	5:	IF NOT bCheckWrappingSen  (* bIConeFeedingPistonEnd *)    THEN  bQAForwardPistonValve:=FALSE;  bAWrappingConvStart1:=TRUE; bAErrorChkBit:=FALSE;
		step:=step+1; END_IF

	6:	IF  InterLockCounter.CV=1 AND bAConeFeedOver   AND NOT bConeMiss2AtWrapConv THEN
		bA2ndConeReached:=TRUE;
		bAWrappingConvStart1:=FALSE;
		step:=step+1;
		END_IF


	7:	IF NOT bAPauseSeq THEN step:=step+1; END_IF

	8:	 step:=step+1;

	9:	 step:=step+1;

	10:	IF  bAutoModeOn AND NOT bQAWrappingConveyorMotor   AND bA2ndConeReached AND InterLockCounter.CV=1 AND NOT bAConeMissErrorAtWrpConv
		AND NOT bConeMiss2AtWrapConv  THEN
		bQAForwardPistonValve:=TRUE;
		 bAErrorChkBit2:=TRUE;
		bAConeFeedOver:=FALSE;
		step:=step+1;
		END_IF

	11:	IF NOT bAPauseSeq THEN step:=step+1; END_IF

	12:	IF  bAutoModeOn AND bIConeFeedingPistonHome  AND bIForwardPistonEnd  AND NOT bAFwdCylRsError  THEN
		(*bQAForwardPistonValve:=FALSE;*)
		bA2ndConeReached:=FALSE;
		(*bAWrappingConvStart2:=TRUE;  *)
		bAFwdPistonComp2:=TRUE;
		step:=step+1;
		END_IF


	13:	 IF NOT bCheckWrappingSen2 (* bIConeFeedingPistonEnd *) THEN  bQAForwardPistonValve:=FALSE;  bAWrappingConvStart2:=TRUE; bAErrorChkBit2:=FALSE;
		step:=step+1; END_IF
(*-=========================mod need here=======================*)
	14:	IF   bIConeFeedingPistonEnd AND  bAConeFeedOver THEN
		bA3rdConeReached:=TRUE;
		bAWrappingConvStart2:=FALSE;
		step:=step+1;
		END_IF


	15:	IF NOT bAPauseSeq THEN step:=step+1; END_IF

	16:	IF  bAutoModeOn AND NOT bQAWrappingConveyorMotor   AND  bA3rdConeReached  AND  InterLockCounter.CV=2   AND bFwdPistonStartTemp  AND NOT bConeMiss1AtWrapConv  THEN
		bQAForwardPistonValve:=TRUE;
		 bAErrorChkBit3:=TRUE;
		bAConeFeedOver:=FALSE;
		step:=step+1;
		END_IF

	17:	IF NOT bAPauseSeq THEN step:=step+1; END_IF

	18:	IF  bAutoModeOn AND bIConeFeedingPistonHome  AND bIForwardPistonEnd  AND NOT bAFwdCylRsError   THEN

	(*	bQAForwardPistonValve:=FALSE; *)
		bA3rdConeReached:=FALSE;
	(*	bAWrappingConvStart3:=TRUE; *)
		bAFwdPistonComp3:=TRUE;
		step:=step+1;
		END_IF


	19:	IF NOT bAPauseSeq THEN step:=step+1; END_IF


	20:	IF NOT bCheckWrappingSen3 (* bIConeFeedingPistonEnd *) THEN  bQAForwardPistonValve:=FALSE;  bAWrappingConvStart3:=TRUE; bAErrorChkBit3:=FALSE;
		step:=step+1; END_IF



	21:	 IF  bAutoModeOn AND bIForwardPistonHome AND   InterLockCounter.CV=3 OR bAByPassOn    THEN
		InterLockCounter.RESET:=TRUE;
		bAWrappingConvStart3:=FALSE;
		step:=step+1;
		END_IF

	22:	IF NOT bAPauseSeq THEN (* InterLockCounter.RESET:=FALSE ;*) bAByPassOn:=FALSE;  step:=0; END_IF



END_CASE


CASE Step12 OF

	0:	IF R_TRIG_5.Q  THEN Step12:=1; TON_5(IN:=FALSE);  bConutEnable:=FALSE ;END_IF

	1:	IF NOT bQAWrappingConveyorMotor THEN Step12:=2;
		ELSE IF InterLockCounter.CV=2 THEN Step12:=2; END_IF END_IF

	2:	IF  TON_5.Q THEN Step12:=3;
		ELSE IF InterLockCounter.CV=2 AND R_TRIG_1.Q  THEN Step12:=3; END_IF  END_IF

	3:	bConutEnable:=TRUE ; Step12:=4;

	4:	Step12:=0;

END_CASE

R_TRIG_1(CLK:= (  bIWrappingConeDeductionSen), Q=> );
R_TRIG_5(CLK:= (  bWrapConvStarted), Q=> );
TON_5(IN:=bIWrappingConeDeductionSen , PT:=t#0.8s , Q=> , ET=> );

(*IF R_TRIG_1.Q (* bIWrappingConeDeductionSen*)  AND bWrapConvStarted THEN bConutEnable:=TRUE ; ELSE bConutEnable:=FALSE ;END_IF *)

InterLockCounter(
	CU:=bConutEnable ,
	RESET:= ,
	PV:= ,
	Q=> ,
	CV=> );

R_TRIG_2(CLK:=bQAWrappingConveyorMotor , Q=> );

IF R_TRIG_2.Q THEN bWrapConvStarted:=TRUE; END_IF


F_TRIG_1(CLK:= bQAWrappingConveyorMotor, Q=> );

IF F_TRIG_1.Q THEN bWrapConvStarted:=FALSE; END_IF
(*Hanging Logic======*)


IF bAErrorChkBit AND bQAForwardPistonValve  AND  bIWrappingConeDeductionSen  THEN bCheckWrappingSen:=TRUE; END_IF

IF  bWrpConvIntOver AND bSealConvIntOver THEN  bAFwdPistonReady:=TRUE; ELSE 	bAFwdPistonReady:=FALSE; END_IF


IF bAErrorChkBit2 AND  bQAForwardPistonValve AND bIWrappingConeDeductionSen AND (  bIWrappingCone1 OR bIWrappingCone2 OR bIWrappingCone3 ) THEN bCheckWrappingSen2:=TRUE; END_IF


IF bAErrorChkBit3 AND  bQAForwardPistonValve AND bIWrappingConeDeductionSen AND   bIWrappingCone1 AND ( bIWrappingCone2 OR bIWrappingCone3 ) THEN bCheckWrappingSen3:=TRUE; END_IF





IF  NOT bIEmergency OR   bAutoModeOff  OR bStopHmi OR bIMCStop  THEN

bAFirstConeReached:=FALSE;
bQAForwardPistonValve:=FALSE;
bAWrappingConvStart1:=FALSE;
bAFwdPistonComp1:=FALSE;
bA2ndConeReached:=FALSE;
step:=0;
bAWrappingConvStart2:=FALSE;
bAFwdPistonComp2:=FALSE;
bA3rdConeReached:=FALSE;
bAWrappingConvStart3:=FALSE;
bAFwdPistonComp3:=FALSE;
bWrpConvIntOver:=FALSE;
bSealConvIntOver:=FALSE;
InterLockCounter.RESET:=TRUE;

ELSE
InterLockCounter.RESET:=FALSE;

END_IF

IF bErrorReset  AND bCheckWrappingSen AND NOT  bIWrappingConeDeductionSen THEN bAErrorChkBit:=FALSE;  bCheckWrappingSen:=FALSE;WrapConeSenDetMes:=''; InterLockCounter.RESET:=TRUE; ELSE InterLockCounter.RESET:=FALSE;END_IF
IF bCheckWrappingSen THEN  WrapConeSenDetMes:='Wrapping Cone Home Sensor Error';END_IF



IF bErrorReset  AND bCheckWrappingSen2 AND NOT  bIWrappingCone1 AND NOT   bIWrappingCone2 AND NOT bIWrappingCone3  THEN bAErrorChkBit2:=FALSE;  bCheckWrappingSen2:=FALSE;WrapConeSenDetMes:=''; END_IF
IF bCheckWrappingSen2 THEN  WrapConeSenDetMes:='Wrapping Cone Sensor Error';END_IF


IF bErrorReset  AND bCheckWrappingSen3 AND NOT   bIWrappingCone2 AND NOT bIWrappingCone3  THEN bAErrorChkBit3:=FALSE;  bCheckWrappingSen3:=FALSE;WrapConeSenDetMes:=''; END_IF
IF bCheckWrappingSen3 THEN  WrapConeSenDetMes:='Wrapping Cone Sensor Error';END_IF
END_PROGRAM

(* POU AutoMode/Wrapping_Unit, ST *)
PROGRAM Wrapping_Unit
VAR

	step1: INT;

	R_TRIG_1: R_TRIG;
	Counter1: CTU;
	WrapConvStartDly: TON;
	WrapR_TRIG_1: R_TRIG;
	bAWrappingConvStartAuto2: BOOL;
	WrapR_TRIG_2: R_TRIG;
	WrapConvStartDly2: TON;
	WrapR_TRIG_3: R_TRIG;
	WrapConvStartDly3: TON;
	bAWrappingConvStartAuto3: BOOL;
	WrapR_TRIG_4: R_TRIG;
	bAWrappingConvStartAuto4: BOOL;
	WrapConvStartDly4: TON;
	WrapR_TRIG_5: R_TRIG;
	bAWrappingConvStartAuto5: BOOL;
	WrapConvStartDly5: TON;
	bAWrapConeCyl1: BOOL;
	bAWrapConeCyl123: BOOL;
	bAWrapConeCyl3: BOOL;
	bAWrapConeCyl23: BOOL;
	bASet1Comp: BOOL;
	bASet2Comp: BOOL;
	bASet: BOOL;
	bASet3Comp: BOOL;
	bA3ConeWrapStarted: BOOL;
	bA6thConeWrapStarted: BOOL;
	bA1ConeWrappOver: BOOL;
	bA2ConeWrappOver: BOOL;
	bAll3ConeWrapOver: BOOL;
	bA5ConeWrappOver: BOOL;
	bA6ConeWrappOver: BOOL;
	bA56ConeWrapOver: BOOL;
	bAWrapConeCyl23_1: BOOL;

	bATemp: BOOL;
	baConv2ndStart: BOOL;
	baConv3rdStart: BOOL;
	baConv4thStart: BOOL;
	baConv5thStart: BOOL;
	bASensorMonitorBit1: BOOL;
	bAWrappingCone123FwdCom: BOOL;
	ni: BOOL;
	step2: INT;
	bAWrappingCone3FwdCom: BOOL;
	step3: INT;
	bAWrappingCone23FwdCom: BOOL;
	step4: INT;
	bAWrappingCone23FwdCom1: BOOL;
	bASet4Comp: BOOL;
	WrapR_TRIG_3_23: R_TRIG;
	bAWrappingConvStartAuto3_23: BOOL;
	WrapConvStartDly3_23: TON;
	bAWrapConeCyl23_1_23: BOOL;
	bAWrappingCone23_23FwdCom1: BOOL;
	WrapR_TRIG_6_23: R_TRIG;
	bAWrappingConvStartAuto4_23: BOOL;
	WrapConvStartDly6_23: TON;
	bIWrappingCone: BOOL;

	bAWrapConeCyl123_23: BOOL;
	bAWrappingCone123_23FwdCom: BOOL;

	step5: INT;
	bAConvRunning1: BOOL;
	bAConvRunning2: BOOL;
	TON_1: TON;
	TON_2: TON;
	bANextLayerStarted: BOOL;
	bAConvStartInterlock: BOOL;
	bAFirstConeAtWrapConv: BOOL;
	baConveyerStarted: BOOL;
	RtrigBit1: BOOL;
	R_TRIG_3: R_TRIG;
	bASensorNok: BOOL;
	WrapConvStartDlyOver: BOOL;
	test: R_TRIG;
	WrappingCone1RT: R_TRIG;
	WrappingConvRT: R_TRIG;
	WCS1Sensed: BOOL;
	TON_3: TON;
	WCS1SenseRst1: BOOL;
	TON_6: TON;
	TON_7: TON;
	TON_8: TON;
	TON_9: TON;
	TON_10: TON;
	TimerStartBit: BOOL;
	bConvRunning: BOOL;
	test1THEN: BOOL;
	test1: BOOL;
	bSaelUnitIntOverTemp: BOOL;
	step6: INT;
	step7: INT;
	bWCSStart3_24: BOOL;
	bStopHmitemp: BOOL;
	bWCSHomeSenOk: BOOL;

	WCSCylsHomeRsErr: BOOL;

	bWCSHomeEndOk: BOOL;
	WCSCylsEndRsErr: BOOL;

	bAWrappingConvStartAuto: BOOL;
	bA3Pushed: BOOL;
	bWCSStart3: BOOL;
	bWCSStart2: BOOL;
	RsChkDly: TON;
	bWrapConvStopped2: BOOL;

	bWrapConvStopped3: BOOL;

	bIWrappingFilmTensionChk1: BOOL;
	bIWrappingFilmTensionChk2: BOOL;
	bIWrappingFilmTensionChk3: BOOL;
	R_TRIG1: F_TRIG;
	R_TRIG2: F_TRIG;
	R_TRIG3: F_TRIG;
	Film1Loaded: BOOL;
	Film3Loaded: BOOL;
	Film2Loaded: BOOL;
	FlimNotLoaded: BOOL;
	FlimChkDly: TON;
	Timer1: TON;
	bAWrapFirstStart: BOOL;
	TON2: TON;
	sSheetNotFeeded: STRING;
	F_TRIG1: F_TRIG;
	F_TRIG2: F_TRIG;
	F_TRIG3: F_TRIG;
	WrappConeBitAlert1: BOOL;
	WrappConeBitAlert2: BOOL;
	WrappConeBitAlert3: BOOL;
	bQAWrappingConveyorMotor1Temp: BOOL;
	checkPolySheet1: BOOL;
	bQAWrappingConveyorMotor2Temp: BOOL;
	Timer6: TON;
	bAllignConeErr1: BOOL;
	bQAWrappingConveyorMotor2Temp2: BOOL;
	checkPolySheet2Temp: BOOL;

	Timer3: TON;
END_VAR
(*========================Wrapping Conveyor Logic in auto Mode=================*)

bQAWrappingConveyorMotor:= (bQAWrappingConveyorMotor1 OR bQAWrappingConveyorMotor2 OR bQAWrappingConveyorMotor3 );

(*===================Wrapping Pinston On/Off Logic In Auto Mode==================*)


bQAWrappingChannelPistonValve1:= (bAWrappingCone123OnAuto  );

bQAWrappingChannelPistonValve2:=( bAWrappingCone123OnAuto );

bQAWrappingChannelPistonValve3:=( bAWrappingCone123OnAuto );


(*========================Wrapping Conveyor  Logic for First Cone in auto Mode =================*)

WrapR_TRIG_1(CLK:=bAWrappingConvStart1  , Q=> );

IF bAutoModeOn AND  WrapR_TRIG_1.Q  THEN  bAWrappingConvStartAuto:=TRUE; END_IF

WrapConvStartDly(IN:= bAWrappingConvStartAuto, PT:=t#0.3s , Q=> , ET=> );

(*=====New Added for Cone Detection At Wrapp Conveyor====*)

IF WrapR_TRIG_1.Q   AND (bIWrappingCone1 OR bIWrappingCone2 OR  bIWrappingCone3 OR bIWrappingConeDeductionSen) THEN WrappConeBitAlert1:=TRUE;ELSE WrappConeBitAlert1:=FALSE;END_IF
IF WrappConeBitAlert1 AND bErrorReset THEN WrappConeBitAlert1:=FALSE; END_IF
IF WrapR_TRIG_2.Q   AND (bIWrappingCone1 OR bIWrappingCone2 OR  bIWrappingCone3 OR bIWrappingConeDeductionSen) THEN WrappConeBitAlert2:=TRUE;ELSE WrappConeBitAlert2:=FALSE;END_IF
IF WrappConeBitAlert2 AND bErrorReset THEN WrappConeBitAlert2:=FALSE; END_IF
IF WrapR_TRIG_3.Q   AND (bIWrappingCone1 OR bIWrappingCone2 OR  bIWrappingCone3 OR bIWrappingConeDeductionSen) THEN WrappConeBitAlert3:=TRUE;ELSE WrappConeBitAlert3:=FALSE;END_IF
IF WrappConeBitAlert3 AND bErrorReset THEN WrappConeBitAlert3:=FALSE; END_IF


IF bAutoModeOn AND  WrapConvStartDly.Q (*AND NOT bCheckWrappingSen  bIWrappingConeDeductionSen *)AND bIWrappingChannelPiston1_Home AND bIWrappingChannelPiston2_Home  AND  bAWrapFirstStart AND bIWrappingChannelPiston3_Home(*  AND NOT bIWrappingCone1 AND NOT bIWrappingCone2 AND NOT bIWrappingCone3 *) AND NOT WrappConeBitAlert1 THEN
bQAWrappingConveyorMotor1:=TRUE;
bAWrapConStart:=FALSE;
bA3ConeWrappOverTemp:=FALSE;
END_IF

    (*==========================  Wrapping Sheet Sensing Error=================*)
(*
IF bQAWrappingConveyorMotor1   THEN
bAErrorChkBit:=TRUE;

IF NOT  bCheckWrappingSen    THEN
bAErrorChkBit:=FALSE;
bQAWrappingConveyorMotor1Temp:=TRUE;
bQAWrappingConveyorMotor1:=FALSE;
END_IF
END_IF
*)



IF   bAutoModeOn AND  bIWrappingConeDeductionSen THEN
bQAWrappingConveyorMotor1:=FALSE;
bQAWrappingConveyorMotor1Temp:=FALSE;
END_IF

(*===============Wrapping Conveyor 2nd  Cone  Logic  in auto Mode==================*)

WrapR_TRIG_2(CLK:= ( bAWrappingConvStart2 ) , Q=> );


IF bAutoModeOn AND  WrapR_TRIG_2.Q THEN  bAWrappingConvStartAuto:=FALSE;  bAWrappingConvStartAuto2:=TRUE; END_IF

WrapConvStartDly2(IN:= bAWrappingConvStartAuto2, PT:=t#0.1s , Q=> , ET=> );


IF bAutoModeOn AND  WrapConvStartDly2.Q  AND bIWrappingChannelPiston1_Home AND bIWrappingChannelPiston2_Home AND bIWrappingChannelPiston3_Home AND bIWrappingConeDeductionSen   AND NOT bAWrapCylRsErrorAuto AND NOT bConeMiss1AtWrapConv AND NOT WrappConeBitAlert2 AND NOT bCheckWrappingSen2  THEN
bQAWrappingConveyorMotor2:=TRUE;

bAConvRunning1:=TRUE;

END_IF
(*
   (*==========================  Wrapping Sheet Sensing Error=================*)
IF bQAWrappingConveyorMotor2 THEN
IF bQAWrappingConveyorMotor2 AND   bIWrappingConeDeductionSen  AND( bIWrappingCone1 OR  bIWrappingCone2 OR  bIWrappingCone3 ) THEN
checkPolySheet2:=TRUE;
checkPolySheet2Temp:=TRUE;
ELSE
checkPolySheet2Temp:=TRUE;

END_IF
END_IF



IF checkPolySheet2Temp AND   bIWrappingConeDeductionSen AND NOT  bIWrappingCone1 AND NOT  bIWrappingCone2 AND NOT  bIWrappingCone3 AND NOT checkPolySheet2   THEN

bQAWrappingConveyorMotor2Temp:=TRUE; bQAWrappingConveyorMotor2:=FALSE;
END_IF

*)
(*
IF bQAWrappingConveyorMotor2Temp THEN Timer6(IN:=TRUE , PT:=t#2s , Q=> , ET=> ); END_IF

IF bQAWrappingConveyorMotor2Temp AND Timer6.Q AND NOT bIWrappingConeDeductionSen THEN bAllignConeErr1:=TRUE;
ELSIF bQAWrappingConveyorMotor2Temp AND Timer6.Q AND  bIWrappingConeDeductionSen THEN bQAWrappingConveyorMotor2Temp2:=TRUE; Timer6(IN:=FALSE);
END_IF
*)



IF  bAutoModeOn AND  bIWrappingCone1 AND   bAConvRunning1    THEN
bWrapConvStopped2:=TRUE;
bWrapConvStopped2Temp:=TRUE;
bQAWrappingConveyorMotor2:=FALSE;
bAWrappingConvStartAuto2:=FALSE;
bAConvRunning1:=FALSE;
END_IF
(*================================== this Logic is for Cone Missing at Cone Detection sensor in wrapping Unit==========================*)
IF bAutoModeOn AND bWrapConvStopped2Temp AND TON2.Q    AND bIWrappingConeDeductionSen THEN bFwdPistonStartTemp:=TRUE; bWrapConvStopped2Temp:=FALSE; END_IF
IF bAutoModeOn AND bWrapConvStopped2Temp THEN   TON2(IN:=TRUE , PT:= t#1s, Q=> , ET=> ); ELSE TON2(IN:=FALSE);
END_IF
IF bAutoModeOn AND TON2.Q AND NOT  bIWrappingConeDeductionSen  THEN  bConeMiss1AtWrapConv:=TRUE; END_IF

IF bAutoModeOn AND bConeMiss1AtWrapConv AND bIWrappingConeDeductionSen AND bErrorReset AND bIWrappingCone1  THEN
bConeMiss1AtWrapConv:=FALSE; TON2(IN:=FALSE); END_IF

(*===============Wrapping Conveyor  3rd Cone  Logic  in auto Mode ==================*)

WrapR_TRIG_3(CLK:=bAWrappingConvStart3 , Q=> );


IF bAutoModeOn AND  WrapR_TRIG_3.Q THEN bAWrappingConvStartAuto3:=TRUE;  checkPolySheet2Temp:=FALSE; bWrapConvStopped2:=FALSE;  END_IF

WrapConvStartDly3(IN:= bAWrappingConvStartAuto3, PT:=t#0.1s , Q=> , ET=> );


IF  bAutoModeOn AND WrapConvStartDly3.Q AND bIWrappingChannelPiston1_Home AND bIWrappingChannelPiston2_Home AND bIWrappingChannelPiston3_Home AND bIWrappingConeDeductionSen AND bIWrappingCone1 AND NOT bAWrapCylRsErrorAuto AND NOT WrappConeBitAlert3  AND NOT bCheckWrappingSen3  AND NOT  bWrapConvStopped2Temp THEN
bQAWrappingConveyorMotor3:=TRUE;
bASensorMonitorBit1:=TRUE;
END_IF

IF   bAutoModeOn AND  bASensorMonitorBit1 AND   bIWrappingCone3 AND NOT bIWrappingConeDeductionSen THEN
bQAWrappingConveyorMotor3:=FALSE;
bAWrappingConvStartAuto3:=FALSE;
bASensorMonitorBit1:=FALSE;
bWrapConvStopped3:=TRUE;
END_IF
(* ================== Cone Missing Logic on Wrapping Conveyor===============*)

IF bWrapConvStopped3 THEN Timer1(IN:=TRUE , PT:=t#1s , Q=> , ET=> ); ELSE  Timer1(IN:=FALSE); END_IF


IF bAutoModeOn AND   Timer1.Q  AND bWrapConvStopped3 AND bIWrappingCone1 AND bIWrappingCone2 AND NOT bConeMiss2AtWrapConv THEN  bAWrapConeCyl123:=TRUE;  bWrapConvStopped3:=FALSE;
ELSIF bAutoModeOn AND Timer1.Q  AND( NOT  bIWrappingCone1 OR NOT bIWrappingCone2  ) THEN bConeMiss2AtWrapConv:=TRUE;
END_IF


(* ==================Error Acknlodge for  Cone Missing Logic on Wrapping Conveyor===============*)


 IF bConeMiss2AtWrapConv AND bAutoModeOn AND bErrorReset AND   bIWrappingCone1 AND  bIWrappingCone2 AND  bIWrappingCone3  THEN bConeMiss2AtWrapConv:=FALSE;  bAByPassOn:=TRUE; END_IF





(*===============Wrapping piston 123 on/off logic  ====================*)
CASE step1 OF

	0:	TON_1(IN:= FALSE);
		step1:=step1+1;

	1:	step1:=step1+1;

	2:	IF bAutoModeOn AND  bAWrapConeCyl123  AND  bIWrappingChannelPiston1_Home   AND bIWrappingChannelPiston2_Home AND bIWrappingChannelPiston3_Home
		  AND ( bWCSStart1 OR bWCSStart2  )  AND SealingOk AND NOT bAWrapwait THEN
		TON_1(IN:= TRUE, PT:=T#0.3s , Q=> , ET=> );
		IF TON_1.Q THEN  step1:=step1+1; END_IF
		END_IF

	3:	bWCSStart1:=FALSE;
		bWCSStart2:=FALSE;
		step1:=step1+1;


	4:	IF bISealingBottomPistonHome AND bISealingTopPistonHome AND  NOT bQASealingConveyorMotor AND NOT bAPauseSeq   AND NOT bASealSepXCylRsError
		AND SealingOk THEN
		bAWrappingCone123OnAuto:=TRUE;
		step1:=step1+1;
		END_IF


	5:	RsChkDly(IN:=FALSE);
		step1:=step1+1;

	6:	IF bAWrappingCone123OnAuto AND bIWrappingChannelPiston1_End AND bIWrappingChannelPiston2_End AND bIWrappingChannelPiston3_End
		AND SealingOk AND bAFilmLoaded   AND NOT bAWrappingCylRsError THEN
		bAConvRunning1:=FALSE;
		bAWrappingCone123FwdCom:=TRUE;
		TON_1(IN:= FALSE);
		step1:=step1+2;
		ELSIF  bAWrappingCone123OnAuto AND bIWrappingChannelPiston1_End AND bIWrappingChannelPiston2_End AND bIWrappingChannelPiston3_End AND NOT bAWrappingCylRsError  AND NOT bAFilmLoaded THEN
		bAFlimNotLoaded:=TRUE;
		bAWrappingCone123OnAuto:=FALSE;
		bAWrapConeCyl123:=FALSE;
		bAPolythinSheetError:=TRUE;
		ConeMissAlarm1:='Sheet NOT Feeded';
		step1:=step1+3;
		ELSIF NOT  bIWrappingChannelPiston1_End OR NOT  bIWrappingChannelPiston2_End OR NOT  bIWrappingChannelPiston3_End  AND  bAWrappingCone123OnAuto   (* AND not  bAFilmLoaded AND NOT bAWrappingCylRsError     *) THEN
		RsChkDly(IN:=TRUE , PT:=t#5s , Q=> , ET=> );
		IF RsChkDly.Q THEN bAWrapCylRsErrorAuto:=TRUE;   bAWrappingCone123OnAuto:=FALSE; step1:=step1+1; END_IF

		END_IF

	7:	IF bErrorReset THEN RsChkDly(IN:=FALSE);
		bAWrapCylRsErrorAuto:=FALSE;
		step1:=4;
		END_IF

	8:	 IF bAWrappingCone123FwdCom AND NOT bAPauseSeq  THEN
		bAWrappingCone123OnAuto:=FALSE;
		bAFilmLoaded:=FALSE;
		step1:=step1+2;
		END_IF

	9:	 IF bFilmErrClear THEN sSheetNotFeeded:='';  bAFlimNotLoaded:=FALSE;bAConvRunning1:=FALSE;
		 step1:=step1+1;END_IF

	10:	bAWrapConeCyl123:=FALSE;
		bA3ConeWrappOverTemp:=TRUE;
		step1:=step1+1;

	11:	bFilmErrClear:=FALSE;step1:=step1+1;

	12:	 IF  bIWrappingChannelPiston1_Home   AND bIWrappingChannelPiston2_Home AND bIWrappingChannelPiston3_Home   THEN
		bAWrappingCone123FwdCom:=FALSE; 		bA3ConeWrappOver:=TRUE;
		bA3Pushed:=TRUE;
		step1:=0;
		END_IF


END_CASE




IF bAWrapConStart OR bA3ConeWrappOverTemp THEN bAWrapFirstStart:=TRUE; ELSE bAWrapFirstStart:=FALSE; END_IF



	(*========================== Wrapping Sheet not Feeded Error==================*)

	IF bAWrappingCone123OnAuto AND  F_TRIG1.Q AND NOT bIWrappingChannelPiston1_End   AND NOT Film1Loaded THEN Film1Loaded:=TRUE;   END_IF

	IF bAWrappingCone123OnAuto AND  F_TRIG2.Q  AND NOT bIWrappingChannelPiston2_End AND NOT Film2Loaded    THEN Film2Loaded:=TRUE;  END_IF

	IF bAWrappingCone123OnAuto AND  F_TRIG3.Q  AND NOT bIWrappingChannelPiston3_End AND NOT Film3Loaded  THEN Film3Loaded:=TRUE;  END_IF


F_TRIG1(CLK:=bIWrappingFilmTensionPlate_1 , Q=> );


F_TRIG2(CLK:=bIWrappingFilmTensionPlate_2, Q=> );
(* IF R_TRIG2.Q THEN Film2Loaded:=TRUE; END_IF *)


F_TRIG3(CLK:=bIWrappingFilmTensionPlate_3 , Q=> );
  (*IF R_TRIG3.Q THEN Film3Loaded:=TRUE; END_IF *)


IF  Film1Loaded AND  Film2Loaded AND  Film3Loaded THEN bAFilmLoaded:=TRUE;   Film1Loaded:=FALSE;  Film2Loaded:=FALSE;  Film3Loaded:=FALSE;  END_IF

R_TRIG1(CLK:= bAWrappingCone123OnAuto , Q=> );

IF R_TRIG1.Q THEN Film1Loaded:=FALSE; Film2Loaded:=FALSE; Film3Loaded:=FALSE;  END_IF


IF bAWrappingCone123OnAuto THEN FlimChkDly(IN:=TRUE , PT:=t#5s , Q=> , ET=> ); ELSE FlimChkDly(IN:=FALSE);   END_IF

IF bAPolythinSheetError AND bErrorReset   THEN  bFilmErrClear:=TRUE; bAPolythinSheetError:=FALSE ; ConeMissAlarm1:=''; END_IF

(*=============== Interlock Logic for  2*3 WCS conveyor===================*)




IF bSaelUnitIntOver THEN
bSaelUnitIntOverTemp:=TRUE;
END_IF



CASE step6 OF


0:	IF bSaelUnitIntOverTemp   THEN                             (*========= need to check for reset Logic=    step6:=0    =======*)
	Step6:=Step6+1;
	END_IF

1:	bWCSStart1:=TRUE;
	bAWrapConStart:=TRUE;

	Step6:=Step6+1;

2:	IF  bASealConvEnd1 THEN
	bSaelUnitIntOverTemp:=FALSE;
	Step6:=Step6+1;
	END_IF

3:	bWCSStart2:=TRUE;
	bASealConvEnd1:=FALSE;
	Step6:=2;


END_CASE

IF NOT  bIEmergency OR  bAutoModeOff  OR bStopHmi  OR bIMCStop  THEN
bAWrappingConvStartAuto:=FALSE;
WrapConvStartDly(IN:=FALSE);
bQAWrappingConveyorMotor1:=FALSE;
bAWrappingConvStartAuto2:=FALSE;
WrapConvStartDly2(IN:=FALSE);
bQAWrappingConveyorMotor2:=FALSE;
bAConvRunning1:=FALSE;
bWrapConvStopped2:=FALSE;
bFwdPistonStartTemp:=FALSE;
bAWrapCylRsErrorAuto :=FALSE;
bConeMiss1AtWrapConv:=FALSE;
bAWrappingConvStartAuto3:=FALSE;
WrapConvStartDly3(IN:=FALSE);
bQAWrappingConveyorMotor3:=FALSE;
bASensorMonitorBit1:=FALSE;
bWrapConvStopped3:=FALSE;
Timer1(IN:=FALSE);
bAWrapConeCyl123:=FALSE;
bConeMiss2AtWrapConv:=FALSE;
step1:=0;
step6:=0;
TON_1(IN:= FALSE);
bAWrappingCone123OnAuto:=FALSE;
bAWrappingCone123FwdCom:=FALSE;
RsChkDly(IN:=FALSE);
bA3ConeWrappOver:=FALSE;
bA3Pushed:=FALSE;
bIWrappingFilmTensionChk1:=FALSE;
bIWrappingFilmTensionChk2:=FALSE;
bIWrappingFilmTensionChk3:=FALSE;

END_IF
END_PROGRAM

(* POU AutoMode/Sealing_Unit, ST *)
PROGRAM Sealing_Unit
VAR
	step: INT;
	tA3ConeStartDly: TON;
	tA3ConeSealCompDly: TON;
	test: BOOL;


END_VAR
IF NOT  bIEmergency   OR bStopHmi  OR  bAutoModeOff  OR bIMCStop THEN
	Step:=0;
	bQASealingSeparatorYAxisPistonValve:=FALSE;
	bQASealingTopPistonValve:=FALSE;
	bQASealingSeparatorXAxisPistonValve:=FALSE;
	bA3ConeWrappOver:=FALSE;
	bMManualSealOn:=FALSE;
	tA3ConeStartDly(IN:=FALSE);
	tA3ConeSealCompDly(IN:=FALSE);

END_IF


CASE step OF

	0:	IF bAutoModeOn  THEN
		Step:=step+1;
		END_IF

	1:	step:=step+1;


	2:	IF bAutoModeOn AND  bA3ConeWrappOver   AND NOT bAPauseSeq  THEN
		tA3ConeStartDly(IN:=TRUE , PT:=t#1.5s , Q=> , ET=> );
		IF tA3ConeStartDly.Q THEN  step:=step+1; END_IF
		END_IF

	3:	step:=step+1;

	4:	IF bAutoModeOn AND   bISealingBottomPistonHome  AND bISealingTopPistonHome AND bISealingSeparatorXAxisHome AND bISealingSeparatorYAxisHome AND  NOT bAPauseSeq THEN
		bQASealingSeparatorYAxisPistonValve:=TRUE;
		bASepYAxisRsErrorChkBit:=TRUE;
		tA3ConeSealCompDly(IN:=FALSE);
		step:=step+1;
		END_IF

	5:	 step:=step+1;

	6:	IF bAutoModeOn AND  bISealingSeparatorYAxisEnd AND  NOT bAPauseSeq  AND NOT bASealSepYCylRsError THEN
		tA3ConeStartDly(IN:=FALSE);
		bQASealingTopPistonValve:=TRUE;
		bASepYAxisRsErrorChkBit:=FALSE;
		step:=step+1;
		END_IF

	7:	step:=step+1;

	8:	IF bAutoModeOn AND  bISealingTopPistonEnd AND bISealingBottomPistonEnd  THEN
		tA3ConeSealCompDly(IN:=TRUE, PT:= SealComDlyTemp, Q=> , ET=> );
		IF tA3ConeSealCompDly.Q THEN   step:=step+1; END_IF
		END_IF

	9:	step:=step+1;

	10:	IF bAutoModeOn AND  bISealingTopPistonEnd AND bISealingBottomPistonEnd (*AND  bISealingSeparatorYAxisEnd*) AND  NOT bAPauseSeq  AND NOT bASealTopBotCylRsError  AND NOT bASealSepYCylRsError  THEN
		bQASealingSeparatorXAxisPistonValve:=TRUE;
		(*bASepYAxisRsErrorChkBit1:=TRUE;  *)
		step:=step+1;
		END_IF

	11:	 bASepYAxisRsErrorChkBit1:=FALSE; step:=step+1;

	12:	IF bAutoModeOn AND  bISealingSeparatorXAxisEnd AND  NOT bAPauseSeq  AND NOT bASealSepXCylRsError THEN

		step:=step+1;
		 END_IF

	13:	 step:=step+1;

	14:	bQASealingTopPistonValve:=FALSE;
		bA3ConeWrappOver:=FALSE;
		bA4thWrappOver:=FALSE;
		bA6thConeWrappOver:=FALSE;
		bA8thConeWrappOver:=FALSE;
		bA6ConeWrappOver23:=FALSE;
		bQASealingSeparatorYAxisPistonValve:=FALSE;
		bQASealingSeparatorXAxisPistonValve:=FALSE;
		step:=step+1;

	15:	step:=step+1;

	16:	IF bAutoModeOn AND  bISealingSeparatorXAxisHome AND  bISealingTopPistonHome AND bISealingBottomPistonHome AND bISealingSeparatorYAxisHome  THEN
		step:=step+1;
		END_IF


	17:	step:=step+1;

	18:	step:=step+1;

	19:	 step:=step+1;

	20:	step:=0;



END_CASE

		IF bAutoModeOn AND NOT bA3ConeWrappOver  AND NOT bA4thWrappOver AND NOT bA6thConeWrappOver AND NOT bA8thConeWrappOver
		 AND  bISealingSeparatorXAxisHome AND  bISealingTopPistonHome AND bISealingBottomPistonHome AND bISealingSeparatorYAxisHome  THEN
		SealingOk:=TRUE; ELSE SealingOk:=FALSE;
		END_IF













































(*

(*================Wrapping Conveyor On/Off Logic==========================*)

CASE step OF
	1:	IF SealDelay.Q   AND NOT bIColumnPushPistonHome THEN
		bQAWrappingConveyorMotor:=TRUE;
		END_IF
	2:	IF bIConeCountSensorVal=3 THEN bQAWrappingConveyorMotor:=FALSE; END_IF

	3: 	IF SealDelay.Q  AND NOT bIColumnPushPistonHome   THEN  bQAWrappingConveyorMotor:=TRUE;	END_IF

	4:	IF bIConeCountSensorVal=1 THEN bQAWrappingConveyorMotor:=FALSE; END_IF

	5:	 IF SealDelay.Q   AND NOT bIColumnPushPistonHome   THEN  bQAWrappingConveyorMotor:=TRUE;	END_IF

	6:	IF bIConeCountSensorVal=2 THEN bQAWrappingConveyorMotor:=FALSE; END_IF


	7:	 IF SealDelay.Q   AND NOT bIColumnPushPistonHome   THEN  bQAWrappingConveyorMotor:=TRUE;	END_IF

	8:	IF bIConeCountSensorVal=2 THEN bQAWrappingConveyorMotor:=FALSE; END_IF


	9:	step:=0;


END_CASE

*)







(*


		IF bAutoModeOn AND  bAWrapConeCyl123 AND bIWrappingChannelPiston1_Home   AND bIWrappingChannelPiston2_Home AND bIWrappingChannelPiston3_Home    THEN
		bAWrappingCone123OnAuto:=TRUE;

		END_IF

		IF  bAutoModeOn AND  bIWrappingChannelPiston1_End AND bIWrappingChannelPiston2_End AND bIWrappingChannelPiston3_End   THEN
		bAWrappingCone123OnAuto:=FALSE;
		bAWrapConeCyl123:=FALSE;


		END_IF

	IF  bAutoModeOn AND  bAWrappingCone123OnAuto  THEN
		bA3ConeWrapStarted:=TRUE;
	END_IF

IF  bA3ConeWrapStarted AND bIWrappingChannelPiston1_End THEN
bA1ConeWrappOver:=TRUE;END_IF

 IF bA3ConeWrapStarted AND bIWrappingChannelPiston2_End THEN
bA2ConeWrappOver:=TRUE;
END_IF

IF bA3ConeWrapStarted AND  bIWrappingChannelPiston3_End THEN
bA3ConeWrappOver:=TRUE;
END_IF


IF bA1ConeWrappOver AND bA2ConeWrappOver AND bA3ConeWrappOver  THEN
bAll3ConeWrapOver:=TRUE;
 bASet1Comp:=TRUE;
END_IF


*)
END_PROGRAM

(* POU AutoMode/Sealing_Conveyor, ST *)
PROGRAM Sealing_Conveyor
VAR

	bA3ConeSealStarted23: BOOL;
	bQASealingConveyor2: BOOL;
	ConvStopDly1_23: TON;
	bA3ConeSealComp23: BOOL;
	step1: INT;
	(*CTU_1: CTU;*)
	bAConeCountSenEnable1: BOOL;
	bA6thConeSealStarted23: BOOL;
	bA6thConeSealComp23: BOOL;
	ConvStopDly2_23: TON;
	step2: INT;
	step3: INT;
	bSealConvIntOverTemp: BOOL;
	bStopHmitemp: BOOL;
	ConeMissErr_1: BOOL;

	ConeMissErr_2: BOOL;
	test: BOOL;
	bA3COneCrossed: BOOL;
	bSealConvStart3: BOOL;
	bSealConvStart1: BOOL;
	TON1: TON;
	Timer1: TON;
	Timer2: TON;

	Timer3: TON;
	bConeMissBit2: BOOL;
	bConeMissBit3: BOOL;
	bConeMissBit1: BOOL;
	Timer4: TON;
	bConeMissBit: BOOL;
	ConeChkDly: TON;
	SealConeMiss: STRING;
	bQASealingConveyor3: BOOL;
	bAConeMissAtSealConv2: BOOL;
	bA3ConeSealComp23Temp: BOOL;
	bTemp: BOOL;

END_VAR
bQASealingConveyorMotor:= bQASealingConveyor1 OR bQASealingConveyor2 OR bQASealingConveyor3 ;


CASE step1 OF

	0:	IF bAutoModeOn  AND   bA3ConeWrappOver AND bQASealingSeparatorYAxisPistonValve  THEN
		CTU_1.RESET:=TRUE;
		TON1(IN:=FALSE);
		bA3ConeSealStarted23:=TRUE;
		ConvStopDly1_23(IN:=FALSE);
		step1:=step1+1;
		END_IF
	1:	IF NOT bAPauseSeq THEN step1:=step1+1; END_IF


	2:	IF bAutoModeOn  AND  bA3ConeSealStarted23 AND bISealingSeparatorXAxisEnd THEN
		bA3ConeSealComp23:=TRUE;
		CTU_1.RESET:=FALSE;
		step1:=step1+1;
		END_IF

	3:	step1:=step1+1;

	4:	IF bAutoModeOn AND   bA3ConeSealComp23Temp  AND   NOT bAPauseSeq    AND NOT bASealSepXCylRsError THEN
		bQASealingConveyor1:=TRUE;
		step1:=step1+1;
		END_IF

	5:	 TON1(IN:=FALSE); step1:=step1+1;


	6:	IF CTU_1.CV>=3 THEN
		bSealConvStart1:=FALSE;
		bSealConvStart3:=FALSE;
		bA3ConeSealComp23Temp:=FALSE;
		bA3ConeSealStarted23:=FALSE;
		bA3COneCrossed:=TRUE;
		TON1(IN:=TRUE, PT:=  t#1s, Q=> , ET=> );
		IF TON1.Q THEN  CTU_1.RESET:=TRUE; step1:=step1+1; END_IF
		END_IF

	7:	bQASealingConveyor1:=FALSE;
		bQASealingConveyor2:=FALSE;
		bQASealingConveyor3:=FALSE;
		bASealConvEnd1:=TRUE;
		CTU_1.RESET:=FALSE;
		TON1(IN:=FALSE);

		step1:=0;



END_CASE

IF NOT bQASealingConveyorMotor AND bIConeCountSensor  THEN bAWrapwait:=TRUE;ELSE bAWrapwait:=FALSE;END_IF

IF bA3ConeSealComp23 THEN  bA3ConeSealComp23Temp:=TRUE;  bA3ConeSealComp23:=FALSE; END_IF


IF bQASealingConveyorMotor AND bIConeCountSensor  THEN
bAConeCountSenEnable1:=TRUE;
ELSE
bAConeCountSenEnable1:=FALSE;
END_IF

CTU_1(
	CU:=bAConeCountSenEnable1 ,
	RESET:= ,
	PV:=3 ,
	Q=> ,
	CV=> );

IF CTU_1.CV<>3 AND (bQASealingConveyor1 OR bQASealingConveyor2 OR bQASealingConveyor3 )THEN
(*ConeMissbit:=TRUE;*)
ConeChkDly(IN:= TRUE , PT:=t#7s , Q=> , ET=> );
ELSE
ConeChkDly(IN:= FALSE);
END_IF


(*
CASE SealingStep OF



	0:	Timer1(IN:=FALSE);
		Timer2(IN:=FALSE);
		Timer3(IN:=FALSE);
		SealingStep:=SealingStep+1;

	1:	IF  ConeMissbit  THEN
		Timer1(IN:=TRUE , PT:=t#2s , Q=> , ET=> );
		IF NOT Timer1.Q  AND (CTU_1.CV ) = 1 THEN SealingStep:=SealingStep+1;
		ELSIF  Timer1.Q	 AND (CTU_1.CV)<>1 THEN  SealingStep:=3;
		END_IF
		END_IF

	2:	IF (CTU_1.CV)=1 THEN
		SealingStep:=SealingStep+2;
		END_IF

	3:	IF  (CTU_1.CV)<>1 THEN
		bConeMissBit1:=TRUE;
		AlarmMessg:='One Cone  Missing From Sealing Conveyor';
		SealingStep:=11;
		ELSIF (CTU_1.CV) = 1  THEN
		AlarmMessg:='';
		SealingStep:=SealingStep+1;
		END_IF


	4:	Timer2(IN:=TRUE , PT:=t#2s , Q=> , ET=> );
		IF NOT Timer2.Q  AND (CTU_1.CV ) = 2 THEN SealingStep:=SealingStep+1;
		ELSIF  Timer2.Q	 AND (CTU_1.CV)<>2 THEN  SealingStep:=6; END_IF


	5:	IF (CTU_1.CV)=2 THEN
		SealingStep:=SealingStep+2; END_IF




	6:	IF  (CTU_1.CV)<>2 THEN
		bConeMissBit2:=TRUE;
		AlarmMessg:='Two Cone  Missing From Sealing Conveyor';
		SealingStep:=11;
		ELSIF (CTU_1.CV) = 2  THEN
		AlarmMessg:='';
		SealingStep:=SealingStep+1;

		END_IF

	7:	Timer3(IN:=TRUE , PT:=t#2s , Q=> , ET=> );
		IF NOT Timer3.Q AND  NOT bAPauseSeq  AND (CTU_1.CV ) =3 THEN SealingStep:=SealingStep+1;
		ELSIF  Timer3.Q AND  NOT bAPauseSeq	 AND (CTU_1.CV)<>3 THEN  SealingStep:=9; END_IF

	8:	IF (CTU_1.CV)=3 THEN
		SealingStep:=10;
		END_IF

	9:	IF (CTU_1.CV) <> 3  THEN
		bConeMissBit3:=TRUE;
		AlarmMessg:='One Cone  Missing From Sealing Conveyor';
		SealingStep:=11;
		ELSIF (CTU_1.CV) = 3  THEN
		AlarmMessg:='';
		SealingStep:=SealingStep+1;
		END_IF


	10:	IF (CTU_1.CV)=0 THEN
		ConeMissbit:=FALSE;
		Timer3(IN:=FALSE);
		Timer2(IN:=FALSE);
		Timer1(IN:=FALSE);
		SealingStep:=0;
		END_IF

	11:	Timer4(IN:=TRUE , PT:= t#3m, Q=> , ET=> );
		IF bConeMissBit  AND  (CTU_1.CV)=1  AND  Timer4.Q THEN(* bAPauseEnable:=TRUE; *)  bQASealingConveyor1:=FALSE;  Step1:=4;  SealingStep:=7;
		ELSIF bConeMissBit  AND  (CTU_1.CV)=2  AND  Timer4.Q THEN (*bAPauseEnable:=TRUE; *) bQASealingConveyor1:=FALSE;  Step1:=4;  SealingStep:=7;
		END_IF

END_CASE




IF bQASealingConveyor1_23 AND CTU_AlarmOnly.CV =3  THEN  bCountLock1:=TRUE; END_IF

IF bQASealingConveyor5_23 AND CTU_AlarmOnly.CV =3  THEN  bCountLock5:=TRUE; END_IF

IF bQASealingConveyor6_23 AND CTU_AlarmOnly.CV =3  THEN  bCountLock6:=TRUE; END_IF


IF bQASealingConveyor2_23 AND CTU_AlarmOnly.CV =6  THEN  bCountLock2:=TRUE; END_IF


IF bQASealingConveyor3_23 AND CTU_AlarmOnly.CV =6  THEN  bCountLock3:=TRUE; END_IF


IF bQASealingConveyor4_23 AND CTU_AlarmOnly.CV =6  THEN  bCountLock4:=TRUE; END_IF


 IF bCountLock1 OR bCountLock2 OR  bCountLock3 OR bCountLock4 OR  bCountLock5 OR bCountLock6 THEN bCountLock:=TRUE; ELSE bCountLock:=FALSE; END_IF
*)


IF bQASealingConveyor1  AND  ConeChkDly.Q   AND   CTU_1.CV<>3  THEN bAConeMissAtSealConv:=TRUE; AlarmMessg:=' Cone  Missing From Sealing Conveyor';  bQASealingConveyor1:=FALSE;  END_IF




IF bAConeMissAtSealConv AND bErrorReset THEN bQASealingConveyor2:=TRUE;  Step1:=5;    AlarmMessg:=''; bAConeMissAtSealConv:=FALSE; END_IF

IF bQASealingConveyor2  AND  ConeChkDly.Q   AND CTU_1.CV<>3   THEN bAConeMissAtSealConv2:=TRUE; AlarmMessg:=' Cone  Missing From Sealing Conveyor';  bQASealingConveyor2:=FALSE;  END_IF

IF bAConeMissAtSealConv2 AND bErrorReset THEN bQASealingConveyor3:=TRUE;  Step1:=5;  ConeChkDly(IN:= FALSE);  AlarmMessg:=''; bAConeMissAtSealConv2:=FALSE; END_IF

IF bQASealingConveyor3 AND ConeChkDly.Q  AND CTU_1.CV<>3 THEN bQASealingConveyor3:=FALSE; bTemp:=TRUE;  AlarmMessg:=' Cone  Missing From Sealing Conveyor'; END_IF

IF bTemp  AND bErrorReset THEN
Step1:=4;  ConeChkDly(IN:= FALSE); bTemp:=FALSE;
END_IF



IF bAConeMissAtSealConv OR bAConeMissAtSealConv2 THEN bAConeMissAtSealConv:=TRUE; ELSE  bAConeMissAtSealConv:=FALSE; END_IF



IF NOT  bIEmergency OR  bAutoModeOff  OR bStopHmi OR bIMCStop  THEN
step1:=0;
bA3ConeSealStarted23:=FALSE;
ConvStopDly1_23(IN:=FALSE);
bA3ConeSealComp23:=FALSE;
bQASealingConveyor1:=FALSE;
bQASealingConveyor2:=FALSE;
bQASealingConveyor3:=FALSE;
bAConeMissAtSealConv:=FALSE;
bAConeMissAtSealConv2:=FALSE;
bAConeMissAtSealConv:=FALSE;
CTU_1.RESET:=TRUE;
bAConeCountSenEnable1:=FALSE;
TON1(IN:=FALSE);
ELSE

CTU_1.RESET:=FALSE;

END_IF
END_PROGRAM

(* POU WeightCalc, ST *)
PROGRAM WeightCalc
VAR
	CounterA: CTU;
	R_TRIG_1: R_TRIG;
	CounterB: CTU;
	R_TRIG_2: R_TRIG;
	R_TRIG_3: R_TRIG;

	ConeCountEnable: BOOL;
	InterLockCounterStartTimer: TON;
	TON_3: TON;
	tResetTiner: TON;
	WCPReadyTemp1: BOOL;
	WCPReadyTemp2: BOOL;
	Det: WORD;
	BreadTemp: BOOL;
	ADSREAD_1: ADSREAD;
	SwithOnButtton: BOOL;
	axis1: BOOL;
	InterLockCounterRESET: BOOL;
	RstStep: INT;
	bStopTiltUnit: BOOL;
	rRetUnitTolMax: REAL;
	rRetUnitTolMin: REAL;
	rRetUnitAWeightok: BOOL;

	TON_4: TON;
	rRetUnitAWeightempt: REAL;
	rRetUnitAWeighttemp: REAL;
	TON_5: TON;
	rRetUnitBWeightok: BOOL;
	TON_6: TON;
	TON_7: TON;
	rGrossWtTolMax: REAL;
	rGrossWtTolMin: REAL;
	TON_8: TON;
	bGrossWieghtOkTemp: BOOL;

	Timer1: TON;
	Timer2: TON;
	bMonitor: BOOL;
	bStartBlinker: BOOL;
	bStartConeFeedConvInBypass: BOOL;
	rRetUnitAWeightNok: BOOL;
	rRetUnitBWeightNok: BOOL;
	iACounterB_PV: INT;
	iACounterA_PV: INT;
	i: INT;

	UnitBWeightBit: BOOL;
	UnitAWeightBit: BOOL;
	weightCheck: INT;
	Timer_3: TON;
	Weight3Move: BOOL;
	var_4: REAL;
	weightCheck1: INT;
	Weight4Move: BOOL;
	Timer_4: TON;
	Weight2Move: BOOL;
	var_2: REAL;
	var_3: REAL;
	Weight1Move: BOOL;
END_VAR
(*===========Reterival unit weight ok and not ok Logic UNIT-A=================*)

(*==== Weight Max & Min Tolerance Setting==========*)

rRetUnitTolMax:= (DFLTNETWT_DIS + NETWTTOL_DIS);

	IF negativetolerance AND bAutoModeOn THEN
	rRetUnitTolMin:= (DFLTNETWT_DIS - NETWTTOL_DIS);
	ELSIF NOT negativetolerance THEN rRetUnitTolMin:= (DFLTNETWT_DIS);
	END_IF
IF rRetUnitAWeight  <= rRetUnitTolMax AND rRetUnitAWeight >=rRetUnitTolMin THEN
rRetUnitAWeightok:=TRUE;
ELSE
rRetUnitAWeightok:=FALSE;
END_IF

IF TON_5.Q   THEN bQAUnitAWeightOkLamp:=TRUE; END_IF


(*
ELSIF Timer1.Q THEN bQAUnitA_LiftPistonValve:=TRUE; ELSE  bQAUnitA_LiftPistonValve:=TRUE; END_IF
IF  bUnitARowStopperStarted  THEN bStartBlinker:=TRUE; ELSE   bStartBlinker:=FALSE;


Timer1(IN:=(bStartBlinker AND NOT Timer2.Q)  , PT:=t#50ms , Q=> , ET=> );

Timer2(IN:=Timer1.Q , PT:=t#50ms , Q=> , ET=> );
*)



(*=========== Unit A Start after wieght ok logic=================*)

IF bIUnitA_StartPB  AND bQAUnitAWeightOkLamp AND bAutoModeOn AND NOT bStartConeFeedConvInBypass THEN  bRetUnitAStart:=TRUE; ELSE bRetUnitAStart:=FALSE;  END_IF





(*============Weight stabilization time======================*)


IF rRetUnitAWeightok THEN TON_4(IN:=TRUE , PT:=t#2s , Q=> , ET=> ); ELSE  TON_4(IN:=FALSE); END_IF

(*============== WEIGHT NOT OK DEFINE TIME ( TON_5)=================*)

IF TON_4.Q THEN TON_5(IN:=TRUE , PT:=t#0.5s , Q=> , ET=> ); ELSE TON_5(IN:=FALSE); END_IF

IF bAutoModeOn AND bIUnitA_RowStopperHome AND NOT rRetUnitAWeightok THEN rRetUnitAWeightNok:=TRUE;  bQAUnitAWeightOkLamp:=FALSE;  ELSE rRetUnitAWeightNok:=FALSE;   END_IF
(*
  IF rRetUnitAWeightNok THEN bRetUnitAStart:=FALSE; END_IF
*)


(*===============weight not ok Indicator on logic====================*)

IF rRetUnitAWeightNok THEN bQAUnitAWeightNokLamp:=TRUE; ELSE  bQAUnitAWeightNokLamp:=FALSE;  END_IF


(*================ Weight ok feedback to Auto Logic=============*)

IF  rRetUnitAWeightok THEN bAUnitAWeighOk:=TRUE;  ELSE bAUnitAWeighOk:=FALSE; END_IF


(*===========Reterival unit weight ok and not ok Logic UNIT-B =================*)



IF rRetUnitBWeight  <= rRetUnitTolMax AND rRetUnitBWeight >=rRetUnitTolMin THEN
rRetUnitBWeightok:=TRUE;
ELSE
rRetUnitBWeightok:=FALSE;
END_IF

IF TON_7.Q THEN bQAUnitBWeightOkLamp:=TRUE; ELSE  bQAUnitBWeightOkLamp:=FALSE;  END_IF




(*=========== Unit B Start after wieght ok logic=================*)

IF bIUnitB_StartPB  AND bQAUnitBWeightOkLamp AND bAutoModeOn  AND NOT bStartConeFeedConvInBypass  THEN  bRetUnitBStart:=TRUE; ELSE bRetUnitBStart:=FALSE; END_IF


(*============Weight stabilization time======================*)


IF rRetUnitBWeightok THEN TON_6(IN:=TRUE , PT:=t#2s , Q=> , ET=> ); ELSE  TON_6(IN:=FALSE); END_IF

(*============== WEIGHT NOT OK DEFINE TIME ( TON_5)=================*)

IF TON_6.Q THEN TON_7(IN:=TRUE , PT:=t#0.5s , Q=> , ET=> ); ELSE TON_7(IN:=FALSE); END_IF

IF bAutoModeOn  AND bIUnitB_RowStopperHome AND NOT rRetUnitBWeightok THEN rRetUnitBWeightNok:=TRUE; ELSE rRetUnitBWeightNok:=FALSE;   END_IF
(*
  IF rRetUnitBWeightNok THEN bRetUnitBStart:=FALSE; END_IF
*)


(*===============weight not ok Indicator on logic====================*)


IF rRetUnitBWeightNok THEN bQAUnitBWeightNokLamp:=TRUE; ELSE  bQAUnitBWeightNokLamp:=FALSE;  END_IF


(*================ Weight ok feedback to Auto Logic=============*)

IF  rRetUnitBWeightok THEN bAUnitBWeighOk:=TRUE; ELSE bAUnitBWeighOk:=FALSE;  END_IF




(*============================================================================================================================================================*)



(*===================UnitA Cone Count Logic================*)

CounterA(
	CU:=bIUnitAConeCrossing ,
	RESET:=R_TRIG_1.Q ,
	PV:=iACounterA_PV ,
	Q=> ,
	CV=> );



(*===================UnitB Cone Count Logic================*)

CounterB(
	CU:=bIUnitBConeCrossing ,
	RESET:=R_TRIG_2.Q ,
	PV:=iACounterB_PV ,
	Q=> ,
	CV=> );





IF bRetUnitAStart AND NOT bRetUnitBStart  (*AND NOT UnitBWeightBit *)THEN UnitAWeightBit:=TRUE; var_1:=rRetUnitAWeight; END_IF
IF bRetUnitBStart AND NOT bRetUnitAStart (*AND NOT UnitAWeightBit*)  THEN UnitBWeightBit:=TRUE; var_2:=rRetUnitBWeight; END_IF

CASE  weightCheck OF


	0:	IF  UnitAWeightBit AND NOT UnitBWeightBit THEN
		Weight1Move:=TRUE;
		weightCheck:=1;END_IF

	1:	IF  Weight1Move AND NOT Weight3Move THEN
		var_3:=var_1;
		Weight3Move:=TRUE;
		Weight1Move:=FALSE;

		weightCheck:=2;END_IF

	2:	IF  CycleComplete AND Weight3Move THEN
		 var_5:=var_3;
		ReportPrint:=TRUE;

		weightCheck:=3;END_IF

	3: 	IF Weight3Move THEN Timer_3(IN:=TRUE , PT:= T#1s , Q=> , ET=> );
		IF Timer_3.Q THEN Weight3Move:=FALSE; UnitAWeightBit:=FALSE;Timer_3(IN:=FALSE);
		weightCheck:=0;END_IF END_IF

END_CASE

CASE  weightCheck1 OF

	0:	IF  UnitBWeightBit AND NOT UnitAWeightBit THEN
		Weight2Move:=TRUE;
		weightCheck1:=1;END_IF

	1:	IF  Weight2Move AND NOT Weight4Move THEN
		var_4:=var_2;
		Weight4Move:=TRUE;
		Weight2Move:=FALSE;

		weightCheck1:=2;END_IF

	2:	IF  CycleComplete1 AND Weight4Move  THEN
		var_5:=var_4;
		ReportPrint:=TRUE;

		weightCheck1:=3;END_IF

	3: 	IF Weight4Move THEN Timer_4(IN:=TRUE , PT:= T#1s , Q=> , ET=> );
		IF Timer_4.Q THEN Weight4Move:=FALSE;UnitBWeightBit:=FALSE; Timer_4(IN:=FALSE);
		weightCheck1:=0;END_IF END_IF

END_CASE


IF  NOT bIEmergency OR   bAutoModeOff  OR bStopHmi OR bIMCStop  THEN

weightCheck1:=0;
weightCheck:=0;
Weight4Move:=FALSE;
Weight2Move:=FALSE;
Weight3Move:=FALSE;
 UnitAWeightBit:=FALSE;
Timer_3(IN:=FALSE);
Weight1Move:=FALSE;
UnitAWeightBit:=FALSE;
UnitBWeightBit:=FALSE;
END_IF
END_PROGRAM

(* POU Startup/INT_All, ST *)
PROGRAM INT_All
VAR
	bCartonOnConv: BOOL;
	bWrpConvIntOverTemp: BOOL;
	bSealConvIntOverTemp: BOOL;
	bAInializeStartedtenp: BOOL;
	bStopInt: BOOL;

	F_TRIG_1: F_TRIG;

END_VAR
IF bInitializeHmi AND bAMcStartInAuto  AND bAutoModeOn (*AND bMCStartInAuto   *) AND NOT   bAInializeStarted    AND NOT bInterlockInitial_2 THEN
bAInitializeSeq:=TRUE;
bAInializeStarted:=TRUE;
bIntialAckBit:=TRUE;
bInterlockInitial_2:=TRUE;
bUnitBReadInt:=TRUE;
END_IF

blink();

WrapConvRst();


SealingConvRst();


SealingUnitRst();



IF  bWrpConvIntOver   AND bSealConvIntOver THEN bAInializeStarted:=FALSE ; bIntialAckBit:=FALSE;END_IF

IF bStopHmi OR bIMCStop  AND bAutoModeOn   THEN bAStop :=TRUE;  bWrpConvIntOver:=FALSE; bSealConvIntOver:=FALSE;  bAMcReady:=FALSE; END_IF

IF( bStopHmi OR bIMCStop)  AND bAutoModeOn AND NOT  bIEmergency THEN bInterlockInitial_2:=FALSE; bUnitBReadInt:=FALSE;END_IF


F_TRIG_1(CLK:= bAInializeStarted, Q=> );

IF F_TRIG_1.Q  AND bAutoModeOn AND   bWrpConvIntOver   AND bSealConvIntOver THEN   bAMcReady:=TRUE; END_IF


IF bAMcReady AND bAutoModeOn AND (bRetUnitAStart OR bRetUnitBStart  ) THEN bAMcRunninig:=TRUE;  bAMcReady:=FALSE; END_IF

(* IF NOT bIEmergency OR bIMCStop   OR bInitializeHmi  THEN bStopInt:=TRUE; ELSE bStopInt:=FALSE; END_IF  *)

(*
AlarmList();
*)


(*
(*=============FULL CARTON CONVEYOR INITIALIZE LOGIC==========*)

	IF    bICartonPosition1 OR  bICartonPosition2 OR  bICartonPosition3  THEN bCartonOnConv:=TRUE; ELSE  bCartonOnConv:=FALSE;  END_IF

	IF 	bAInitializeSeq  AND  bCartonOnConv   AND bAutoModeOn  THEN
	sCartonConvStatus:='Clear the Cone on Carton Conveyor';
	ELSIF 	bAInitializeSeq AND NOT bCartonOnConv AND bAutoModeOn THEN
	bClearConeInt:=TRUE;
	bCartonOnConv:=FALSE;
	sCartonConvStatus:='';
	END_IF
*)
END_PROGRAM

(* POU Startup/blink, CFC *)
PROGRAM blink
VAR
	timer1: TON;
	timer2: TON;
END_VAR
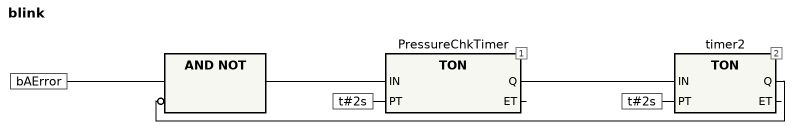
_CFC_ (* Continuous Function Chart, elements in execution order *)
#0 AND NOT(bAError, NOT #2.Q)
#1 PressureChkTimer:TON(IN: #0, PT: t#2s)
#2 timer2:TON(IN: #1.Q, PT: t#2s)
_END_CFC_
END_PROGRAM

(* POU Startup/WrapConvRst, ST *)
PROGRAM WrapConvRst
VAR
	step: INT;
	bConeAtWrppingConveyor1: BOOL;
	TON_1: TON;
	bConePresent: BOOL;
	bAResetHmitemp: BOOL;

	ConeOnWrapConveyAck: BOOL;
END_VAR
IF NOT  bIEmergency OR bStopHmi  OR bAutoModeOff OR bIMCStop  THEN
		bQAWrappingConveyorMotor1:=FALSE;
		bQAWrappingConveyorMotor2:=FALSE;
		bQAWrappingConveyorMotor3:=FALSE;
		bQMWrappingConveyorMotor:=FALSE;
		ConeOnWrapConveyAck:=FALSE;
		bQRWrappingConveyorMotor:=FALSE;
		TON_1(IN:=FALSE);
		bConePresent:=FALSE; step:=0; bAInializeStarted:=FALSE ;
		bQGross_Roller_On:=FALSE;
		bQGross_Cylinder_On:=FALSE;
END_IF





CASE step OF

	0:	 IF bSaelUnitIntOver AND bAutoModeOn THEN
		bQAWrappingConveyorMotor1:=FALSE;
		bQAWrappingConveyorMotor2:=FALSE;
		bQAWrappingConveyorMotor3:=FALSE;
		bQMWrappingConveyorMotor:=FALSE;
		ConeOnWrapConveyAck:=TRUE;
		TON_1(IN:=FALSE);
		step:=step+1;
		END_IF

	1:	bQRWrappingConveyorMotor:=TRUE;
		bSaelUnitIntOver:=FALSE;
		step:=step+1;

	2:	TON_1(IN:=TRUE , PT:=T#10s , Q=> , ET=> );
		IF TON_1.Q THEN
		step:=step+1;
		END_IF

	3:	IF TON_1.Q AND  bQWrappingConveyorMotor AND bConePresent THEN
		step:=step+1;
		ELSIF  TON_1.Q AND  bQWrappingConveyorMotor AND NOT bConePresent THEN
		step:=step+2;
		END_IF

	4:	bQRWrappingConveyorMotor:=FALSE;
		TON_1(IN:=FALSE);
		sWrapConvStatus:='Clear Cone At Wapping Conveyor';
		bConePresent:=FALSE;
		step:=step+1;

	5:	IF NOT bConePresent AND bAutoModeOn   THEN
		TON_1(IN:=FALSE);
		bQRWrappingConveyorMotor:=FALSE;
		sWrapConvStatus:=' ';
		step:=step+1;
		END_IF

	6:	TON_1(IN:=FALSE);
		bWrpConvIntOver:=TRUE;
		ConeOnWrapConveyAck:=FALSE;
		step:=0;

END_CASE


	IF  bAInializeStarted AND (bIWrappingCone1 OR bIWrappingCone2 OR bIWrappingCone3  OR  bIWrappingConeDeductionSen )  AND bAutoModeOn AND ConeOnWrapConveyAck THEN
	bConePresent:=TRUE;
	END_IF

	IF bConePresent  THEN
	ConeMissAlarm:='Allign the Cone at  Wrapping Conveyer ';
	ELSE
	ConeMissAlarm:='No Cone ON Wrapping Conveyer';
	END_IF

	IF  bAInializeStarted AND NOT bIWrappingCone1 AND NOT  bIWrappingCone2 AND NOT  bIWrappingCone3  AND NOT  bIWrappingConeDeductionSen   AND bAutoModeOn AND ConeOnWrapConveyAck
	THEN bConePresent:=FALSE;
	END_IF
END_PROGRAM

(* POU Startup/SealingConvRst, ST *)
PROGRAM SealingConvRst
VAR
	step: INT;
	bConeAtWrppingConveyor1: BOOL;
	TON_1: TON;
	bConePresent: BOOL;
	TON_1Running: BOOL;

END_VAR
CASE step OF

	0:	 IF bSaelUnitIntOver AND bAutoModeOn THEN
		bQASealingConveyorMotor:=FALSE;
		bQMSealingConveyorMotor:=FALSE;
		bQASealingConveyor1:=FALSE;
		step:=step+1;
		END_IF

	1:	bQRSealingConveyorMotor:=TRUE;
		bSaelUnitIntOver:=FALSE;
		step:=step+1;

	2:	IF bConePresent THEN
		step:=step+2;
		ELSIF NOT bConePresent THEN
		step:=step+1;
		END_IF

	3:	IF  TON_1Running  AND bConePresent THEN
		step:=step+1;
		ELSIF TON_1.Q  AND NOT bConePresent THEN
		step:=step+2;
		END_IF

	4:	bQRSealingConveyorMotor:=FALSE;
		TON_1(IN:=FALSE);
		sSealConvStatus:='Clear Cone At Sealing Conveyor';
		bConePresent:=FALSE;
		step:=step+1;

	5:	IF NOT bConePresent AND bAutoModeOn   THEN
		sSealConvStatus:=' ';
		bQRSealingConveyorMotor:=FALSE;
		step:=step+1;
		END_IF

	6:	TON_1(IN:=FALSE);
		bSealConvIntOver:=TRUE;
		step:=0;

END_CASE


(*
IF  bIColumnconeDetection  THEN
bConePresent:=TRUE;
ELSE
bConePresent:=FALSE;
END_IF

*)



IF TON_1.ET >t#1ms AND  TON_1.ET<=t#10s THEN
TON_1Running:=TRUE;
ELSE
TON_1Running:=FALSE;
END_IF



TON_1(IN:=bQRSealingConveyorMotor , PT:=T#10s , Q=> , ET=> );
END_PROGRAM

(* POU Startup/SealingUnitRst, ST *)
PROGRAM SealingUnitRst
VAR
	bARWrappingCone123FwdCom: BOOL;
	TON_1: TON;
	step: INT;
	tA3ConesealStartDly: TON;
	tA3ConeSealCompDly: TON;

	bFwdRevPistonRst: BOOL;

END_VAR
IF NOT  bIEmergency   OR bStopHmi  OR  bAutoModeOff  OR bIMCStop THEN
bInitializeHmi:=FALSE;
bAInitializeSeq:=FALSE;
bQMWrappingChannelPistonValve1:=FALSE;
bQMWrappingChannelPistonValve2:=FALSE;
bQMWrappingChannelPistonValve3:=FALSE;
bQMForwardPistonValve:=FALSE;
bAWrappingCone123OnAuto:=FALSE; bARWrappingCone123FwdCom:=FALSE; bARWrappingCone123OnRst:=FALSE;
bQAForwardPistonValve:=FALSE;
bQMForwardPistonValve:=FALSE;
bFwdPistonRst:=FALSE;
tA3ConeSealCompDly(IN:=FALSE);
bASepYAxisRsErrorChkBit1:=FALSE; bA3ConeWrappOver:=FALSE; tA3ConesealStartDly(IN:=FALSE); bAR3ConeWrappOver:=FALSE;
bQRSealingSeparatorYAxisPistonValve:=FALSE; step:=0;
bQRSealingSeparatorXAxisPistonValve:=FALSE;
bQRSealingTopPistonValve:=FALSE;
END_IF

bQRWrappingChannelPistonValve1:=bARWrappingCone123OnRst;
bQRWrappingChannelPistonValve2:=bARWrappingCone123OnRst;
bQRWrappingChannelPistonValve3:=bARWrappingCone123OnRst;


CASE step OF

	0:	IF  bAutoModeOn AND bAInitializeSeq THEN
		bInitializeHmi:=FALSE;
		Step:=step+1;
		END_IF


	1:	bQMWrappingChannelPistonValve1:=FALSE;
		bQMWrappingChannelPistonValve2:=FALSE;
		bQMWrappingChannelPistonValve3:=FALSE;
		bQMForwardPistonValve:=FALSE;
		bAWrappingCone123OnAuto:=FALSE;
		bQAForwardPistonValve:=FALSE;
		bQMForwardPistonValve:=FALSE;
		bAInitializeSeq:=FALSE;
		Step:=step+1;


	2:	sMessage:='Check Cylinder top & Bottom';  IF NOT bQASealingConveyorMotor AND bISealingSeparatorXAxisHome AND  bISealingTopPistonHome AND bISealingBottomPistonHome
		AND bISealingSeparatorYAxisHome THEN
		bFwdPistonRst:=TRUE;
		bARWrappingCone123OnRst:=TRUE;
		step:=step+1; sMessage:='';
		END_IF


	3:	IF bARWrappingCone123OnRst AND bIWrappingChannelPiston1_End AND bIWrappingChannelPiston2_End AND bIWrappingChannelPiston3_End THEN
		bARWrappingCone123FwdCom:=TRUE;
		TON_1(IN:= FALSE);
		step:=step+1;
		END_IF

	4:	 IF bARWrappingCone123FwdCom THEN
		bARWrappingCone123OnRst:=FALSE;
		step:=step+1;
		END_IF

	5:	 IF  bIWrappingChannelPiston1_Home   AND bIWrappingChannelPiston2_Home AND bIWrappingChannelPiston3_Home   THEN bAR3ConeWrappOver:=TRUE;
		step:=step+1; END_IF


	6:	IF bAutoModeOn AND  bAR3ConeWrappOver  THEN
		tA3ConesealStartDly(IN:=TRUE , PT:=t#2s , Q=> , ET=> );
		IF tA3ConesealStartDly.Q THEN  step:=step+1; END_IF
		END_IF

	7:	IF bAutoModeOn AND   bISealingBottomPistonHome  AND bISealingTopPistonHome AND bISealingSeparatorXAxisHome AND bISealingSeparatorYAxisHome   THEN
		bQRSealingSeparatorYAxisPistonValve:=TRUE;
		tA3ConeSealCompDly(IN:=FALSE);
		bASepYAxisRsErrorChkBit1:=TRUE;
		  step:=step+1;
		END_IF

	8:	IF bAutoModeOn AND  bISealingSeparatorYAxisEnd  AND NOT bASealSepYCylRsError  THEN
		tA3ConesealStartDly(IN:=FALSE);
		bQRSealingTopPistonValve:=TRUE;
		bASepYAxisRsErrorChkBit1:=FALSE;
		step:=step+1;
		END_IF

	9:	IF bAutoModeOn AND  bISealingTopPistonEnd AND bISealingBottomPistonEnd AND NOT bASealBotCylRsError AND NOT bASealTopCylRsError  THEN
		tA3ConeSealCompDly(IN:=TRUE, PT:= t#2s, Q=> , ET=> );
		IF tA3ConeSealCompDly.Q THEN   step:=step+1; END_IF
		END_IF


	10:	IF bAutoModeOn AND  bISealingTopPistonEnd AND bISealingBottomPistonEnd AND bISealingSeparatorYAxisEnd THEN
		bQRSealingSeparatorXAxisPistonValve:=TRUE;
		step:=step+1;
		END_IF



	11:	IF bAutoModeOn AND  bISealingSeparatorXAxisEnd  AND NOT bASealSepXCylRsError THEN
		step:=step+1;
		 END_IF

	12:	bQRSealingTopPistonValve:=FALSE;
		bA3ConeWrappOver:=FALSE;
		bQRSealingSeparatorYAxisPistonValve:=FALSE;
		bQRSealingSeparatorXAxisPistonValve:=FALSE;
		step:=step+1;

	13:	IF bAutoModeOn AND  bISealingSeparatorXAxisHome AND  bISealingTopPistonHome AND bISealingBottomPistonHome AND bISealingSeparatorYAxisHome  THEN

		step:=step+1;
		END_IF

	14:	bSaelUnitIntOver:=TRUE;
		step:=step+1;



	15:	step:=0;



END_CASE

IF bFwdPistonRst THEN bQRForwardPistonValve:=TRUE;  END_IF

IF bIForwardPistonEnd  THEN bFwdPistonRst:=FALSE;  bFwdRevPistonRst:=FALSE; bQRForwardPistonValve:=FALSE;  END_IF
END_PROGRAM

(* POU New Folder/Cylinder_Alarm, ST *)
PROGRAM Cylinder_Alarm
VAR
	RS_Error_1:RS_Error;
	RS_Error_2:RS_Error;
	RS_Error_3:RS_Error;
	RS_Error_4:RS_Error;
	RS_Error_5:RS_Error;
	RS_Error_6:RS_Error;
	RS_Error_7:RS_Error;
	RS_Error_8:RS_Error;
	RS_Error_9:RS_Error;


	BlinkTimer1: TON;
	BlinkTimer2: TON;
	RS_Error_10: RS_Error;
	bASepYAxisRsErrorChkOut: BOOL;
	TON_1: TON;
	bBlinkStart: BOOL;
	bAErrortemp: BOOL;
END_VAR
(*===============All Alarms============*)

IF bAConeFeedCylRsError OR   bPloySheetSensError OR bAFwdCylRsError OR bAWrappingCylRsError OR  bASupplyPressureError OR bAPolythinSheetError OR  ConeAlignErr OR bASealTopBotCylRsError OR bASealSepXCylRsError OR bASealSepYCylRsError
 OR bAConeMissAtSealConv  OR bAEmergencyPressed OR bCheckWrappingSen  OR bCheckWrappingSen2 OR bCheckWrappingSen3  OR bGrossWieghtNOk  OR bGrossWtCylEndSenError THEN bAError :=TRUE; ELSE  bAError:=FALSE; END_IF

(*=======Blinker ==============*)
(*
IF bAError AND NOT BlinkTimer2.Q THEN bBlinkStart:=TRUE; ELSE  bBlinkStart:=FALSE; END_IF

BlinkTimer1(IN:=bBlinkStart , PT:=t#2s , Q=> , ET=> );

BlinkTimer2(IN:=BlinkTimer1.Q , PT:=t#5s , Q=> , ET=> );
*)
(*============ Buzzer on/Off logic============*)

IF    bAError THEN bABuzzer :=TRUE; ELSE bABuzzer:=FALSE; END_IF
IF bAError THEN
sAlarmStatus:='   Alarms Occured. Go To Active Alarms';
ELSE
sAlarmStatus:=' No Alarms ';
END_IF

(*.....................Emergency Alarm................................*)

IF NOT bIEmergency THEN bAEmergencyPressed:=TRUE; ELSE bAEmergencyPressed:=FALSE; END_IF

IF bAEmergencyPressed (*AND BlinkTimer1.Q *)THEN bEmPopUp:=TRUE; ELSE bEmPopUp:=FALSE; END_IF

(*Emg*)
IF NOT  bIEmergency   OR bStopHmi  OR  bAutoModeOff  OR bIMCStop THEN
	bAConeFeedCylRsError:=FALSE;
	bAWrappingCylRs1Error:=FALSE;
	bAWrappingCylRs2Error:=FALSE;
	bAWrappingCylRs3Error:=FALSE;
	bAFwdCylRsError:=FALSE;
	bASealBotCylRsError:=FALSE;
	bASealTopCylRsError:=FALSE;
	bASealSepXCylRsError:=FALSE;
	bASealSepYCylRsError:=FALSE;  bASepYAxisRsErrorChkBit1:=FALSE;  bASepYAxisRsErrorChkBit:=FALSE;   bASepYAxisRsErrorChkOut:=FALSE;
	bAReset_all_error:=TRUE;
ELSE bAReset_all_error:=FALSE;


 END_IF

(*......................................Cone Feeding Piston Alarm.............................*)




RS_Error_1(
	bValveOutOn:=bQAConeFeedingPistonValve ,
	bReedSwithIn:=bIConeFeedingPistonEnd ,
	bErroReset:= (bErrorReset OR bAReset_all_error),
	sMsgIn:= ,
	RS_ErrChkDly:=t#5s ,
	bRsError=>bAConeFeedCylRsError ,
	sMsgOut=> );

IF RS_Error_1.bRsError THEN
RS_Error_1.sMsgIn:='Cone Feeding Piston End Sensor Timeout Error' ;
ELSE
RS_Error_1.sMsgIn:='Continue Machine Operation' ;
END_IF
HMIFeedPiston:=RS_Error_1.sMsgIn;


(*......................................Wrapping Channel Piston1 Alarm.............................*)


RS_Error_2(
	bValveOutOn:=bQWrappingChannelPistonValve1(*bAWrapCylRsErrorAuto*),
	bReedSwithIn:=bIWrappingChannelPiston1_End,
	bErroReset:=(bErrorReset OR bAReset_all_error),
	sMsgIn:= ,
	RS_ErrChkDly:=t#5s ,
	bRsError=> bAWrappingCylRs1Error ,
	sMsgOut=> );
IF  RS_Error_2.bRsError  THEN
RS_Error_2.sMsgIn:=' Wrapping  Piston1 End Sensor Timeout Error' ;

ELSE
RS_Error_2.sMsgIn:='Continue Machine Operation' ;

END_IF

HMIWrapPiston1:=RS_Error_2.sMsgIn;


IF bErrorReset THEN   bAWrapCylRsErrorAuto :=FALSE; END_IF


(*......................................Wrapping Channel Piston2 Alarm.............................*)

RS_Error_3(
	bValveOutOn:=bQWrappingChannelPistonValve2,
	bReedSwithIn:=bIWrappingChannelPiston2_End,
	bErroReset:=(bErrorReset OR bAReset_all_error),
	sMsgIn:= ,
	RS_ErrChkDly:=t#5s ,
	bRsError=> bAWrappingCylRs2Error,
	sMsgOut=> );

IF  RS_Error_3.bRsError  THEN
RS_Error_3.sMsgIn:=' Wrapping  Piston2 End Sensor Timeout Error' ;


ELSE
RS_Error_3.sMsgIn:='Continue Machine Operation' ;
END_IF

HMIWrapPiston2:=RS_Error_3.sMsgIn;

(*......................................Wrapping Channel Piston3 Alarm.............................*)


RS_Error_4(
	bValveOutOn:=bQWrappingChannelPistonValve3,
	bReedSwithIn:=bIWrappingChannelPiston3_End,
	bErroReset:=(bErrorReset OR bAReset_all_error) ,
	sMsgIn:= ,
	RS_ErrChkDly:=t#5s ,
	bRsError=>bAWrappingCylRs3Error ,
	sMsgOut=> );

IF RS_Error_4.bRsError THEN
RS_Error_4.sMsgIn:=' Wrapping  Piston3 End Sensor Timeout Error' ;

ELSE
RS_Error_4.sMsgIn:='Continue Machine Operation' ;
END_IF

HMIWrapPiston3:=RS_Error_4.sMsgIn;

IF bAWrappingCylRs1Error OR bAWrappingCylRs2Error OR bAWrappingCylRs3Error THEN bAWrappingCylRsError:=TRUE; ELSE bAWrappingCylRsError:=FALSE; END_IF
IF bErrorReset THEN   bAWrappingCylRsError :=FALSE; END_IF




(*.................................Cone Forward Piston Alarm............................................*)

RS_Error_5(
	bValveOutOn:=bQForwardPistonValve,
	bReedSwithIn:=bIForwardPistonEnd,
	bErroReset:=(bErrorReset OR bAReset_all_error) ,
	sMsgIn:= ,
	RS_ErrChkDly:=t#5s ,
	bRsError=>bAFwdCylRsError ,
	sMsgOut=> );
IF  RS_Error_5.bRsError THEN
RS_Error_5.sMsgIn:=' Forward Piston End Sensor Timeout Error';
ELSE
RS_Error_5.sMsgIn:='Continue Machine Operation' ;
END_IF

HMIForwdPiston:=RS_Error_5.sMsgIn;

(*.................................Sealing Bottom Piston Alarm............................................*)

RS_Error_6(
	bValveOutOn:=bQSealingTopPistonValve,
	bReedSwithIn:=bISealingBottomPistonEnd,
	bErroReset:=(bErrorReset OR bAReset_all_error) ,
	sMsgIn:= ,
	RS_ErrChkDly:=t#5s ,
	bRsError=> bASealBotCylRsError,
	sMsgOut=> );
IF RS_Error_6.bRsError THEN
RS_Error_6.sMsgIn:='Sealing Bottom Piston End Sensor Timeout Error';
ELSE
RS_Error_6.sMsgIn:='Continue Machine Operation' ;
END_IF

HMISealBotPiston:=RS_Error_6.sMsgIn;

(*.................................Sealing Top Piston Alarm............................................*)

RS_Error_7(
	bValveOutOn:=bQSealingTopPistonValve,
	bReedSwithIn:=bISealingTopPistonEnd,
	bErroReset:=(bErrorReset OR bAReset_all_error) ,
	sMsgIn:= ,
	RS_ErrChkDly:=t#4s ,
	bRsError=>bASealTopCylRsError ,
	sMsgOut=> );
IF  RS_Error_7.bRsError THEN
RS_Error_7.sMsgIn:='Sealing Top Piston End Sensor Timeout Error';
ELSE
RS_Error_7.sMsgIn:='Continue Machine Operation' ;
END_IF

HMISealTopPiston:=RS_Error_7.sMsgIn;

IF bASealBotCylRsError OR bASealTopCylRsError THEN bASealTopBotCylRsError:=TRUE; ELSE bASealTopBotCylRsError:=FALSE; END_IF




(*.................................Sealing Seperator X Axis  Alarm............................................*)

RS_Error_8(
	bValveOutOn:=bQSealingSeparatorXAxisPistonValve,
	bReedSwithIn:=bISealingSeparatorXAxisEnd,
	bErroReset:=(bErrorReset OR bAReset_all_error) ,
	sMsgIn:= ,
	RS_ErrChkDly:=t#8s ,
	bRsError=>bASealSepXCylRsError ,
	sMsgOut=> );
IF RS_Error_8.bRsError THEN
RS_Error_8.sMsgIn:=' X- Axis Piston End Sensor Timeout Error';
ELSE
RS_Error_8.sMsgIn:='Continue Machine Operation' ;
END_IF
HmiXAxisPiston:=RS_Error_8.sMsgIn;

(*.................................Sealing Seperator Y Axis  Alarm...........................................*)

IF bASepYAxisRsErrorChkBit1 OR bASepYAxisRsErrorChkBit THEN bASepYAxisRsErrorChkOut:=TRUE; ELSE bASepYAxisRsErrorChkOut:=FALSE; END_IF

RS_Error_9(
	bValveOutOn:=bASepYAxisRsErrorChkOut ,
	bReedSwithIn:=bISealingSeparatorYAxisEnd,
	bErroReset:=(bErrorReset OR bAReset_all_error) ,
	sMsgIn:= ,
	RS_ErrChkDly:=t#5s ,
	bRsError=>bASealSepYCylRsError ,
	sMsgOut=> );
IF RS_Error_9.bRsError THEN
RS_Error_9.sMsgIn:=' Y-Axis Piston End Sensor Timeout Error';
ELSE
RS_Error_9.sMsgIn:='Continue Machine Operation' ;
END_IF
HmiYAxisPiston:=RS_Error_9.sMsgIn;



(*.................................Supply Pressure  Alarm...........................................*)
(*
RS_Error_10(
	bValveOutOn:=bAutoModeOn,
	bReedSwithIn:=bIPressureSwitch,
	bErroReset:=bErrorReset ,
	sMsgIn:= ,
	RS_ErrChkDly:=t#10s ,
	bRsError=>bASupplyPressureError ,
	sMsgOut=> );
IF RS_Error_10.bRsError THEN
RS_Error_10.sMsgIn:=' Supply Pressure Timeout Error';
ELSE
RS_Error_10.sMsgIn:='Continue Machine Operation' ;
END_IF
HmiSupplyPressureMsg:=RS_Error_10.sMsgIn;


*)
IF bAutoModeOn AND NOT bIPressureSwitch THEN TON_1(IN:= TRUE, PT:= t#10s , Q=> , ET=> ); END_IF

IF bAutoModeOn AND TON_1.Q THEN bASupplyPressureError:=TRUE; END_IF

IF bAutoModeOn AND bASupplyPressureError AND bIPressureSwitch  THEN bASupplyPressureError:=FALSE;  TON_1(IN:= FALSE);  END_IF

IF bASupplyPressureError AND BlinkTimer1.Q THEN bPrssurePopUp:=TRUE; ELSE bPrssurePopUp:=FALSE; END_IF
END_PROGRAM

(* POU FunctionBlocks/RS_Error, ST *)
FUNCTION_BLOCK RS_Error
VAR_INPUT
	bValveOutOn: BOOL;
	bReedSwithIn: BOOL;
	bErroReset: BOOL;
	sMsgIn: STRING;
	RS_ErrChkDly: TIME;
END_VAR
VAR_OUTPUT
	bRsError: BOOL;
	sMsgOut: STRING;
END_VAR
VAR
	FbStep: INT;
	Timer1: TON;
END_VAR
CASE FbStep OF


	0:	Timer1(IN:=FALSE);  FbStep:=FbStep+1;

	1:	IF bValveOutOn THEN FbStep:=FbStep+1; END_IF

	2:	IF bValveOutOn THEN  Timer1(IN:=TRUE , PT:=RS_ErrChkDly , Q=> , ET=> );
		IF Timer1.Q THEN FbStep:=FbStep+1; ;END_IF
		ELSE
		Timer1(IN:=FALSE);  FbStep:= 0 ;
		END_IF


	3:	IF bReedSwithIn THEN  FbStep:=FbStep+1;
		ELSIF NOT bReedSwithIn THEN FbStep:=FbStep+2; END_IF

	4:	IF  NOT bValveOutOn THEN sMsgOut:='';  FbStep:=0; END_IF

	5:	bRsError:=TRUE;  sMsgOut:=sMsgIn; FbStep:=FbStep+1;

	6:	IF bReedSwithIn AND  bErroReset  THEN bRsError:=FALSE; sMsgOut:='' ;  FbStep:=0;
		ELSIF NOT   bReedSwithIn AND    bErroReset THEN bRsError:=FALSE;   sMsgOut:='' ;   FbStep:=0;
		 END_IF

END_CASE
END_FUNCTION_BLOCK

(* POU New Folder/ConeAllignAlarm, ST *)
PROGRAM ConeAllignAlarm
VAR
	ConeMiss: INT;
	TON_1: TON;
	TON_2: TON;
	ConeMissErr: RS_Error;
	TON1: TON;

	bPloyShoeetSensError: BOOL;
END_VAR
(*...................Cone Allignment Alarm.....................*)

IF bQAWrappingConveyorMotor1 THEN TON1(IN:=TRUE , PT:= t#5s, Q=> , ET=> );  ELSE  TON1(IN:=FALSE); END_IF
IF TON1.Q AND NOT bIWrappingConeDeductionSen THEN bAConeMissErrorAtWrpConv:=TRUE; END_IF
IF TON1.Q  AND bIWrappingConeDeductionSen THEN bAConeMissErrorAtWrpConv:=FALSE; ConeMissAlarm:='';  TON1(IN:=FALSE);END_IF
IF bErrorReset THEN TON1(IN:=FALSE); END_IF

IF NOT bIEmergency OR bStopHmi THEN bAConeMissErrorAtWrpConv:=FALSE; END_IF



IF bAConeMissErrorAtWrpConv THEN
ConeMissAlarm:='Allign the Cone At  Wrapping Conveyer';
ELSIF bConeMiss1AtWrapConv THEN
ConeMissAlarm:='Allign the Cone At Wrapping Conveyer ';
ELSIF bConeMiss2AtWrapConv THEN
ConeMissAlarm:='Allign the Cone At  Wrapping Conveyer ';
ELSIF bPloySheetSensError THEN
ConeMissAlarm:='Allign the Cone At  Wrapping Conveyer ';
ELSIF NOT bAConeMissErrorAtWrpConv AND NOT bConeMiss1AtWrapConv AND NOT bConeMiss2AtWrapConv  AND NOT bPloySheetSensError THEN
ConeMissAlarm:=' ';

END_IF


IF  bConeMiss1AtWrapConv OR bConeMiss2AtWrapConv OR  bAConeMissErrorAtWrpConv  THEN ConeAlignErr:=TRUE; ELSE  ConeAlignErr:=FALSE; END_IF
IF bAConeMissErrorAtWrpConv AND bErrorReset THEN bAConeMissErrorAtWrpConv:=FALSE;END_IF
END_PROGRAM

(* POU New Folder/ConeMiss_Alarm, ST *)
PROGRAM ConeMiss_Alarm
VAR
	FeedForward: INT;

	iSensorOnVal: UINT;
END_VAR
(*CASE ConeMiss OF
	0: IF UnitASenSelet=14 OR UnitASenSelet=13 OR UnitASenSelet= 11 OR UnitASenSelet= 7 THEN
	CountMess:=' Cone  NOT Missing';
	ConeMiss:=ConeMiss+1;
	END_IF

	1: IF UnitASenSelet=14 OR UnitASenSelet=13 OR UnitASenSelet= 11 OR UnitASenSelet= 7 THEN
	CountMess:='One Cone Missing';
	ConeMiss:=ConeMiss+1;
	END_IF

	2: IF UnitASenSelet=12 OR UnitASenSelet=10 OR UnitASenSelet= 9 OR UnitASenSelet= 6 OR UnitASenSelet= 5 OR UnitASenSelet= 3 THEN
	CountMess:='Two Cone Missing';
	ConeMiss:=ConeMiss+1;
	END_IF
END_CASE
*)

;
END_PROGRAM

(* POU Common, ST *)
PROGRAM Common
VAR
	F_TRIG_1: F_TRIG;
	R_TRIG_1: R_TRIG;
	bAllAutoOutOff: BOOL;
	bManModeOn: BOOL;
	bManModeOff: BOOL;
	F_TRIG_2: F_TRIG;
	EverRunTimer: TON;

	sSecond: STRING;
	sMinute: STRING;
	sHour: STRING;
	sTIMEtemp2: STRING;
	sTIMEtemp1: STRING;
	sTIMETemp3: STRING;
	wTodayToHmiFinal: STRING;

	wTodayToHmi_Report: STRING;
	sBagNoRep1: STRING;
	sBagNo: INT;

	cartonno:INT;
	sBagNo1: BOOL;
	sBagNo2: BOOL;
	sBagNo3: BOOL;
	sBagNo4: BOOL;
	sBagNo5: BOOL;
	sDayFDate: STRING;
	sMonthFDate: STRING;
	sDayMonthDate: STRING;

	sDateRepo: STRING;

END_VAR
	F_TRIG_1(CLK:=bIAutoManual , Q=> );

	R_TRIG_1(CLK:=bManualModeOn , Q=> );


IF F_TRIG_1.Q THEN bAutoModeOff:=TRUE; END_IF


IF R_TRIG_1.Q THEN bManModeOn:=TRUE; END_IF


IF bAutoModeOff AND bManModeOn THEN bAllAutoOutOff:=TRUE; bAutoModeOff:=FALSE; bManModeOn:=FALSE;  END_IF

 (*  IF bManualModeOn THEN bAutoModeOff:=FALSE; bManModeOn:=FALSE; END_IF  *)

IF biResetPb OR bErrorResethmi THEN bErrorReset:=TRUE;
ELSE bErrorReset:=FALSE; END_IF


	F_TRIG_2(CLK:=bManualModeOn , Q=> );


IF F_TRIG_2.Q THEN bAllAutoOutOff:=FALSE; END_IF



(*=============Company Logo Popup Window appear logic=============*)
PopUp:=TRUE;

EverRunTimer(IN:=PopUp , PT:=t#5s , Q=> , ET=> );

(*==============Negative Tolerance Enable Hmi===================*)


IF bNegTolEnableHMI THEN NegToleranceEnabled:=TRUE; END_IF

IF bNegTolDisableHMI THEN NegToleranceEnabled:=FALSE; END_IF


(*======================= RTC==============================*)

(*FB_DateTime_1(NET_ID:='s ' , Date_Time=> );*)

DateTimeVar:=FB_DateTime_1.Date_Time;

(*===== Current Date to Hmi and Reports=========*)


wTodayToHmi:=MID(STR:=DateTimeVar, LEN:=10, POS:=1);
wTodayToHmiFinal:=MID(STR:=DateTimeVar, LEN:=20, POS:=1);

sDATEFinal:=  (wTodayToHmiFinal);
(*=======Current TIME to Reports========*)
sTIME:= CONCAT (sTIMETemp3, sSecond) ;
sTIMETemp3:=CONCAT(sTIMEtemp2, ':');

sTIMEtemp2:=CONCAT( sTIMEtemp1 , sMinute);

sTIMEtemp1:=CONCAT(sHour, ':');

sHour:=DWORD_TO_STRING(FB_DateTime_1.FBLTIME.systemTime.wHour);

sMinute:=DWORD_TO_STRING(FB_DateTime_1.FBLTIME.systemTime.wMinute);

sSecond:=DWORD_TO_STRING(FB_DateTime_1.FBLTIME.systemTime.wSecond);

(*wTodayToHmi:=STRING_TO_WORD(wTodayToHmiTemp);  *)

logDay:= WORD_TO_STRING (FB_DateTime_1.FBLTIME.systemTime.wDay);

FB_DateTime_1.FBLTIME.systemTime.wDayOfWeek;

FB_DateTime_1.FBLTIME.systemTime.wHour;

FB_DateTime_1.FBLTIME.systemTime.wMilliseconds;


FB_DateTime_1.FBLTIME.systemTime.wMinute;

LogMonth:= WORD_TO_STRING (FB_DateTime_1.FBLTIME.systemTime.wMonth);



FB_DateTime_1.FBLTIME.systemTime.wSecond;



LogYear:=WORD_TO_STRING (FB_DateTime_1.FBLTIME.systemTime.wYear);










					(****************DATE AND TIME***********)

(*======================= RTC==============================*)

FB_DateTime_2(NET_ID:='5.69.203.190.1.1 ' , Date_Time=> );

IF FB_DateTime_1.FBLTIME.systemTime.wHour >0 AND  FB_DateTime_1.FBLTIME.systemTime.wHour<9 THEN sHourPreFix:='0';

sHou:=CONCAT(STR1:=sHourPreFix, Str2:=WORD_TO_STRING(FB_DateTime_1.FBLTIME.systemTime.wHour));

ELSIF FB_DateTime_1.FBLTIME.systemTime.wHour >=10 AND  FB_DateTime_1.FBLTIME.systemTime.wHour<=24 THEN

sHou:=WORD_TO_STRING(FB_DateTime_1.FBLTIME.systemTime.wHour);

END_IF




IF FB_DateTime_1.FBLTIME.systemTime.wDay >0 AND  FB_DateTime_1.FBLTIME.systemTime.wDay<10 THEN sDayPreFix:='0';

sDay:=CONCAT(STR1:=sDayPreFix, Str2:=WORD_TO_STRING(FB_DateTime_1.FBLTIME.systemTime.wDay));

ELSIF FB_DateTime_1.FBLTIME.systemTime.wDay >=10 AND  FB_DateTime_1.FBLTIME.systemTime.wDay<=31 THEN

sDay:=WORD_TO_STRING(FB_DateTime_1.FBLTIME.systemTime.wDay);

END_IF




IF FB_DateTime_1.FBLTIME.systemTime.wMonth >0 AND  FB_DateTime_1.FBLTIME.systemTime.wMonth<10 THEN sMonthPreFix:='0';

sMonth:=CONCAT(STR1:=sMonthPreFix, Str2:=WORD_TO_STRING(FB_DateTime_1.FBLTIME.systemTime.wMonth));

ELSIF FB_DateTime_1.FBLTIME.systemTime.wMonth >=10 AND  FB_DateTime_1.FBLTIME.systemTime.wMonth<=12 THEN

sMonth:=WORD_TO_STRING(FB_DateTime_1.FBLTIME.systemTime.wMonth);

END_IF
cartonno:=((*CartonNoHmi*)DINT_TO_INT(CARTONNO_DIS));


IF cartonno>=0 AND cartonno<10 THEN sBagNo1:=TRUE;sBagNo2:=FALSE;sBagNo3:=FALSE;sBagNo4:=FALSE;sBagNo5:=FALSE;
ELSIF cartonno >= 10 AND cartonno < 100 THEN sBagNo2:=TRUE;sBagNo1:=FALSE;sBagNo3:=FALSE;sBagNo4:=FALSE;sBagNo5:=FALSE;
ELSIF cartonno >= 100 AND cartonno < 1000 THEN sBagNo3:=TRUE;sBagNo2:=FALSE;sBagNo1:=FALSE;sBagNo4:=FALSE;sBagNo5:=FALSE;
ELSIF cartonno >= 1000 AND cartonno < 10000 THEN sBagNo4:=TRUE;sBagNo2:=FALSE;sBagNo3:=FALSE;sBagNo1:=FALSE;sBagNo5:=FALSE;
ELSIF cartonno >= 10000 THEN sBagNo5:=TRUE;sBagNo2:=FALSE;sBagNo3:=FALSE;sBagNo4:=FALSE;sBagNo1:=FALSE;END_IF
IF sBagNo1 THEN sBagNoRep1:='0000';
ELSIF sBagNo2 THEN sBagNoRep1:='000';
ELSIF sBagNo3 THEN sBagNoRep1:='00';
ELSIF sBagNo4 THEN sBagNoRep1:='0';
ELSIF sBagNo1 THEN sBagNoRep1:='';
END_IF


sBagNoRep:=CONCAT(STR1:=(sBagNoRep1), STR2:=DINT_TO_STRING(CARTONNO_DIS));



sDayF1:=CONCAT(STR1:=sDay, STR2:=':');
sMonthF1:=CONCAT(STR1:=sMonth, STR2:=':');
sDayMonth1:=CONCAT(STR1:=sDayF1, STR2:=sMonthF1);
sDayMonthYear1:=CONCAT(STR1:=sDayMonth1, STR2:=WORD_TO_STRING(FB_DateTime_1.FBLTIME.systemTime.wYear));




sDayFDate:=CONCAT(STR1:=sDay, STR2:='/');
sMonthFDate:=CONCAT(STR1:=sMonth, STR2:='/');
sDayMonthDate:=CONCAT(STR1:=sDayFDate, STR2:=sMonthFDate);
sDayMonthYearDate:=CONCAT(STR1:=sDayMonthDate, STR2:=(*WORD_TO_STRING(FB_DateTime_1.FBLTIME.systemTime.wYear)*)sDateRepo);


sDateRepo:=MID(STR:=WORD_TO_STRING(FB_DateTime_1.FBLTIME.systemTime.wYear), LEN:=2, POS:=3);

sDaateReport:=(sDayMonthYearDate);




sDayF:=CONCAT(STR1:=sDay, STR2:='_');
sMonthF:=CONCAT(STR1:=sMonth, STR2:='_');
sDayMonth:=CONCAT(STR1:=sDayF, STR2:=sMonthF);
sDayMonthYear:=CONCAT(STR1:=sDayMonth, STR2:=WORD_TO_STRING(FB_DateTime_1.FBLTIME.systemTime.wYear));

ReportPath:=CONCAT(STR1:='ProductionData', STR2:='_');
ReportPath_Final:=CONCAT(STR1:=ReportPath, STR2:=sDayMonthYear);

ReportPath_Final_1:=CONCAT(STR1:='\\ACP\Reports\', STR2:=ReportPath_Final);
ReportPath_Final_2:=CONCAT(STR1:=ReportPath_Final_1, STR2:='.csv');
END_PROGRAM

(* POU AutoMode/DataLog_1, ST *)
PROGRAM DataLog_1
VAR
	stStation1_ProductionData:Production_Data;
	ST1_ProductionDataValues: STRING(3000);
	S1_iCyc_Count_DISP: INT;
	S1_iACT_HLD_TIMEDISP: INT;
	stActiveuserCredential: BOOL;
	nPressureMaxvalue: REAL;
	OperatorName: STRING;
	nMinimumTopTempLimit_ST1: INT;
	nMaximumTopTempLimit_ST1: INT;
	nTOPTempMaxvalue: UINT;
	nMinimumBTMTempLimit_ST1: INT;
	nBTMTempMaxvalue: UINT;
	nMaximumBTMTempLimit_ST1: INT;
	Set_HLDTIME: INT;
	S_1_iPressure: REAL;
	rS_PressureRange1: REAL;
	nMaxEnergy: REAL;
	nMaxPower: REAL;
	S_iSET_COUNT: INT;
	S1_iTotCyc_Count_DISP: INT;
	sJobStatus_ST1: STRING;
	sStation1_ProductionData_FileName: STRING(80) := 'Hard Disk\Reports\Test1\ProductionData.csv';
	Fb_LoagProductionData: DATA_LOG_Save;
	SaveData: BOOL;
	ST1_ProductionData: STRING(500);
	Fb_CreateFileFormat_1: Fb_CreateFileFormat;
	bEnableFileFormat: BOOL;
	wTodayTemp: STRING;
	sDateTemp: STRING;
	sOLDFileName_ST1: T_MaxString;
	Fb_FormatDrive_1: Fb_FormatDrive;
	bFileDelete: BOOL;
	Fb_CopyBackupAL_Server_LogOf_1: Fb_CopyFileToRemotePC;
	bool2: BOOL;
	bAstart: BOOL;
	TON_1: TON;
	TON_2: TON;
	CTU_1: CTU;
	R_TRIG_1: R_TRIG;
	R_TRIG_2: R_TRIG;
	bACreateNewFile: BOOL;
	ReportStep: INT;
	bANewDay: BOOL;
	Timer1: TON;
	Timer2: TON;
	R_TRIG1: R_TRIG;


	iUnitBNetWtTemp1: REAL;
	rRetUnitBWeightTemp1: REAL;
	StepTemp1: INT;
	rRetUnitBWeightTemp2: REAL;
	StepTemp2: INT;
	BCreateDir: BOOL;
	FB_CreateDir_1: FB_CreateDir;
	bANewDaytemp: BOOL;
	bit2: BOOL;
	hfile: UINT;
	FB_FileOpen_1: FB_FileOpen;
	test: BOOL;
	bit3: BOOL;
	FB_FileWrite_1: FB_FileWrite;
	bEnableFileFormattemp: BOOL;
	BDelete: BOOL;
	FB_FileDelete_1: FB_FileDelete;
	Timer3: TON;
	iCartoNoHmiTemp: DWORD;
	dateInint: WORD;
	E_OpenPath: E_OpenPath;
	FB_FileDelete_2: FB_FileDelete;
	btest: BOOL;
	iLotNoPrevious: STRING;
	CartonNo:INT;
	SameLotNo:BOOL;


	TON_CountCheck: TON;

	LotChangeCompleted: BOOL;
END_VAR
;(*FileCreateTemp;

Fb_CreateFileFormat_1(
	sInputMessage:=ST1_ProductionData ,
	sFileName:='ProductionData' ,
	sDirectory:='\\Admin-PC\Public\' (*  'Hard Disk\Reports\Indo\'  *),
	bEnable:=bEnableFileFormat ,
	wToday:=wTodayTemp ,
	sDate=> sDateTemp,
	bNewDateFound=> bANewDay,
	sOldFileName=>sOLDFileName_ST1 ,
	sFilePathFinal=> );

FB_FileDelete_2(
	sNetId:='192.168.0.103.1.1' ,
	sPathName:= sStation1_ProductionData_FileName ,
	ePath:=E_OpenPath ,
	bExecute:=bFileDelete ,
	tTimeout:=t#1s ,
	bBusy=> ,
	bError=> ,
	nErrId=> );

IF bAutoModeOn THEN Pgm_NoHmi:=1; END_IF
(*bLoadPgm;
IF (bloadRecipeHmi OR bSaveRecipeHmi) THEN
iCartoNoHmiTemp:=iCartoNoHmi;
ELSE
iCartoNoHmiTemp:=(ITotalSample +iCartoNoHmi);
END_IF

iCartonSample:=iCartoNoHmiTemp;*)

		stStation1_ProductionData.S_No						:=INT_TO_STRING( Pgm_NoHmi );
		stStation1_ProductionData.ConeType				:=INT_TO_STRING( iATotalNoOfCones );
		stStation1_ProductionData.CartonNo					:=INT_TO_STRING(CurrentCartonNo)(*CartonNoHmi*);
		stStation1_ProductionData.LotNo					:= (iLotNoHmi);
		stStation1_ProductionData.SDateF					:= (sDATEFinal);
		stStation1_ProductionData.NetWt					:=REAL_TO_STRING(var_5);
		stStation1_ProductionData.WorkOrderNo				:= (iWorkOrderNoHmi);
		stStation1_ProductionData.DefaultNettWeight			:=REAL_TO_STRING (DefaultNetWeightHmi);
		stStation1_ProductionData.DefaultGrossWeight		:= REAL_TO_STRING(DefaultGrossWeightHmi);
		stStation1_ProductionData.Blend					:= (BlendHmi);
		stStation1_ProductionData.Shade					:= (ShadeHmi );
		stStation1_ProductionData.ConeTip					:= (ConeTipHmi);
		stStation1_ProductionData.ConeNettWeight			:= (*REAL_TO_STRING*)(ConeNettHmi);
		stStation1_ProductionData.ConeLength				:=REAL_TO_STRING (ConeLengthHmi);
		stStation1_ProductionData.Dom_Exp					:= (Dom_ExpHmi);
		stStation1_ProductionData.PackType				:= (PackTypeHmi);
		stStation1_ProductionData.CountCode				:= (CountCodeHmi);




		(*	######## LOG PRODUCTION DATA		#####	*)

ST1_ProductionDataValues:= CONCAT(stStation1_ProductionData.S_No,',');
ST1_ProductionDataValues:=	 CONCAT( ST1_ProductionDataValues,stStation1_ProductionData.ConeType);
ST1_ProductionDataValues:= CONCAT( ST1_ProductionDataValues,',');
ST1_ProductionDataValues:=	 CONCAT( ST1_ProductionDataValues,stStation1_ProductionData.CartonNo);
ST1_ProductionDataValues:= CONCAT( ST1_ProductionDataValues,',');
ST1_ProductionDataValues:=	 CONCAT( ST1_ProductionDataValues,stStation1_ProductionData.LotNo);
ST1_ProductionDataValues:= CONCAT( ST1_ProductionDataValues,',');
(*ST1_ProductionDataValues:=	 CONCAT( ST1_ProductionDataValues,stStation1_ProductionData.ActualNetWt	);
ST1_ProductionDataValues:= CONCAT( ST1_ProductionDataValues,',');*)
ST1_ProductionDataValues:=	 CONCAT( ST1_ProductionDataValues,stStation1_ProductionData.SDateF);
ST1_ProductionDataValues:= CONCAT( ST1_ProductionDataValues,',');
ST1_ProductionDataValues:=	 CONCAT( ST1_ProductionDataValues,stStation1_ProductionData.NetWt);
(*ST1_ProductionDataValues:= CONCAT( ST1_ProductionDataValues,',');
ST1_ProductionDataValues:=	 CONCAT( ST1_ProductionDataValues,stStation1_ProductionData. NetWt );
ST1_ProductionDataValues:= CONCAT( ST1_ProductionDataValues,',');
ST1_ProductionDataValues:=	 CONCAT( ST1_ProductionDataValues,stStation1_ProductionData.StandardGrossWt);
ST1_ProductionDataValues:= CONCAT( ST1_ProductionDataValues,',');
ST1_ProductionDataValues:=	 CONCAT( ST1_ProductionDataValues,stStation1_ProductionData.sEmpConeWt);*)
ST1_ProductionDataValues:= CONCAT( ST1_ProductionDataValues,',');    (**)
ST1_ProductionDataValues:=	 CONCAT( ST1_ProductionDataValues,stStation1_ProductionData.WorkOrderNo);
ST1_ProductionDataValues:= CONCAT( ST1_ProductionDataValues,',');

ST1_ProductionDataValues:=	 CONCAT( ST1_ProductionDataValues,stStation1_ProductionData.DefaultNettWeight);
ST1_ProductionDataValues:= CONCAT( ST1_ProductionDataValues,',');
ST1_ProductionDataValues:=	 CONCAT( ST1_ProductionDataValues,stStation1_ProductionData.DefaultGrossWeight);
ST1_ProductionDataValues:= CONCAT( ST1_ProductionDataValues,',');
ST1_ProductionDataValues:=	 CONCAT( ST1_ProductionDataValues,stStation1_ProductionData.Blend);
ST1_ProductionDataValues:= CONCAT( ST1_ProductionDataValues,',');
ST1_ProductionDataValues:=	 CONCAT( ST1_ProductionDataValues,stStation1_ProductionData.Shade);
ST1_ProductionDataValues:= CONCAT( ST1_ProductionDataValues,',');
ST1_ProductionDataValues:=	 CONCAT( ST1_ProductionDataValues,stStation1_ProductionData.ConeTip);
ST1_ProductionDataValues:= CONCAT( ST1_ProductionDataValues,',');
ST1_ProductionDataValues:=	 CONCAT( ST1_ProductionDataValues,stStation1_ProductionData.ConeNettWeight);
ST1_ProductionDataValues:= CONCAT( ST1_ProductionDataValues,',');
ST1_ProductionDataValues:=	 CONCAT( ST1_ProductionDataValues,stStation1_ProductionData.ConeLength);
ST1_ProductionDataValues:= CONCAT( ST1_ProductionDataValues,',');
ST1_ProductionDataValues:=	 CONCAT( ST1_ProductionDataValues,stStation1_ProductionData.Dom_Exp);
ST1_ProductionDataValues:= CONCAT( ST1_ProductionDataValues,',');
ST1_ProductionDataValues:=	 CONCAT( ST1_ProductionDataValues,stStation1_ProductionData.PackType);
ST1_ProductionDataValues:= CONCAT( ST1_ProductionDataValues,',');
ST1_ProductionDataValues:=	 CONCAT( ST1_ProductionDataValues,stStation1_ProductionData.CountCode);
ST1_ProductionDataValues:= CONCAT( ST1_ProductionDataValues,'$0A');
(*==========Saving the Data to Report===========*)


sStation1_ProductionData_FileName:= Fb_CreateFileFormat_1.sOldFileName ; (*    'Hard Disk\Reports\Test1\ProductionData.csv' ;*)


Fb_LoagProductionData(
	bStartDataLog:= SaveData ,
	sDataLogFileName:=sStation1_ProductionData_FileName ,
	LogData:=ST1_ProductionDataValues ,
	bErrorDataLog=> );






(*=============== file copy from CX Controller to Remote PC & File Delete In CX Device======================*)


	Fb_CopyBackupAL_Server_LogOf_1(
		bMakeDirectory:= ,
		bCopyFile:=bool2,
		sDestDriveName:=' \\Admin-PC\Public\',
		sSourceDirectory:='\Hard Disk\Reports\Indo' ,
		 );

(*\\ramrajg-nb2\Ramaraj_public\   *)

  (*Hard Disk\Reports\  *)

Fb_FormatDrive_1(sDriveName:= '\\Admin-PC\Public\', bFormatDisk:=bFileDelete );


CASE ReportStep OF

	0:	 IF R_TRIG1.Q   THEN  FileCreateTemp:=TRUE; Timer3(IN:=FALSE); ReportStep:=1; END_IF

	1:	(*		##### Station 1 Production Data	#####	*)

		ST1_ProductionData:= CONCAT( 'S.No',',');
		ST1_ProductionData:=	 CONCAT( ST1_ProductionData,'Cone Type');
		ST1_ProductionData:= CONCAT( ST1_ProductionData,',');
		ST1_ProductionData:=	 CONCAT( ST1_ProductionData,'Carton No');
		ST1_ProductionData:= CONCAT( ST1_ProductionData,',');
		ST1_ProductionData:=	 CONCAT( ST1_ProductionData,'Lot No');
		ST1_ProductionData:= CONCAT( ST1_ProductionData,',');
		ST1_ProductionData:=	 CONCAT( ST1_ProductionData,'Date');
		ST1_ProductionData:= CONCAT( ST1_ProductionData,',');
		ST1_ProductionData:=	 CONCAT( ST1_ProductionData,'Net Weight');
		ST1_ProductionData:= CONCAT( ST1_ProductionData,',');
		ST1_ProductionData:=	 CONCAT( ST1_ProductionData,'Work Order No');
		ST1_ProductionData:= CONCAT( ST1_ProductionData,',');

ST1_ProductionData:=	 CONCAT( ST1_ProductionData,'Default Net Weight');
		ST1_ProductionData:= CONCAT( ST1_ProductionData,',');
ST1_ProductionData:=	 CONCAT( ST1_ProductionData,'Defaulr Gross Weight');
		ST1_ProductionData:= CONCAT( ST1_ProductionData,',');
ST1_ProductionData:=	 CONCAT( ST1_ProductionData,'Blend');
		ST1_ProductionData:= CONCAT( ST1_ProductionData,',');
ST1_ProductionData:=	 CONCAT( ST1_ProductionData,'Shade');
		ST1_ProductionData:= CONCAT( ST1_ProductionData,',');
ST1_ProductionData:=	 CONCAT( ST1_ProductionData,'Cone Tip');
		ST1_ProductionData:= CONCAT( ST1_ProductionData,',');
ST1_ProductionData:=	 CONCAT( ST1_ProductionData,'Cone Nett Weight');
		ST1_ProductionData:= CONCAT( ST1_ProductionData,',');
ST1_ProductionData:=	 CONCAT( ST1_ProductionData,'Cone Length');
		ST1_ProductionData:= CONCAT( ST1_ProductionData,',');
ST1_ProductionData:=	 CONCAT( ST1_ProductionData,'Dom Exp');
		ST1_ProductionData:= CONCAT( ST1_ProductionData,',');
ST1_ProductionData:=	 CONCAT( ST1_ProductionData,'Pack Type');
		ST1_ProductionData:=CONCAT( ST1_ProductionData,',');
ST1_ProductionData:=	 CONCAT( ST1_ProductionData,'CountCode');
		ST1_ProductionData:= CONCAT( ST1_ProductionData,'$0A');
		ReportStep:=2;

	2:	Timer1(IN:=FALSE);
		bANewDay:=FALSE;
		ReportStep:=3;


	3:	bEnableFileFormat:=TRUE;
		Timer1(IN:=TRUE , PT:=T#100ms , Q=> , ET=> );
		IF Timer1.Q THEN bEnableFileFormat:=FALSE;  ReportStep:=4; END_IF


	4:
		SaveData:=TRUE;
		Timer1(IN:=FALSE);
		ReportStep:=5;

	5:	Timer3(IN:=TRUE , PT:=T#10s , Q=> , ET=> );
		IF Timer3.Q THEN SaveData:=FALSE;bFileDelete:=TRUE;  ReportStep:=6; END_IF

	6:	 bFileDelete:=FALSE;Timer3(IN:=FALSE); FileCreateTemp:=FALSE; ReportStep:=0;

END_CASE



R_TRIG1(CLK:=CycleComplete OR CycleComplete1 , Q=> );

IF ParametesSave THEN LotNoChange:=TRUE;ELSE LotNoChange:=FALSE;END_IF

IF bAutoModeOn AND bAPauseSeq AND   LotNoChange  THEN
	CurrentCartonNo:=CartonNoHmi;LotChangeCompleted:=FALSE;SameLotNo:=FALSE;
 END_IF

IF bAutoModeOn AND LotChangeCompleted THEN
	iLotNoPrevious:=iLotNoHmi;
END_IF



IF iLotNoPrevious=iLotNoHmi THEN SameLotNo:=TRUE;
ELSE SameLotNo:=FALSE;END_IF

CASE CartonNo OF

0: 	IF (CycleComplete OR CycleComplete1) THEN CartonNo:=CartonNo+1;TON_CountCheck(IN:=FALSE);END_IF

1:	IF SameLotNo THEN CartonNo:=CartonNo+1;
	ELSIF NOT SameLotNo THEN CartonNo:=3;END_IF

2:	CurrentCartonNo:=CurrentCartonNo+1;CartonNo:=4;

3:	CurrentCartonNo:=CartonNoHmi;CartonNo:=CartonNo+1;

4:	TON_CountCheck(IN:=TRUE, PT:=t#30s, Q=> , ET=> );
	IF TON_CountCheck.Q THEN CartonNo:=CartonNo+1;END_IF

5:	CartonNo:=0;LotChangeCompleted:=TRUE;

END_CASE









(*
CASE StepTemp1 OF
	0:	IF bRetUnitBStart THEN rRetUnitBWeightTemp1:=rRetUnitBWeight; StepTemp1:=StepTemp1+1; END_IF

	1:	IF UnitBCompleteCheckCount.CV = 18 AND bAutoModeOn THEN rRetUnitBWeightTemp2:=rRetUnitBWeightTemp1;  StepTemp1:=0; END_IF
 END_CASE




CASE StepTemp2 OF
	0:	IF bRetUnitBStart THEN rRetUnitBWeightTemp1:=rRetUnitBWeight; StepTemp2:=StepTemp2+1; END_IF

	1:	IF c18_ConeCounter1.CV = 18 AND bAutoModeOn THEN rRetUnitBWeightTemp2:=rRetUnitBWeightTemp1; c18_ConeCounter1.RESET:=TRUE;  StepTemp2:=StepTemp2+1; END_IF

	2:	c18_ConeCounter1.RESET:=FALSE;  StepTemp2:=0;
 END_CASE*)


(*IF LotAHmi AND NOT LotBHmi AND NOT LotCHmi THEN LotASelected:=TRUE;LotBSelected:=FALSE;LotCSelected:=FALSE;END_IF
IF NOT LotAHmi AND  LotBHmi AND NOT LotCHmi THEN LotBSelected:=TRUE;LotASelected:=FALSE;LotCSelected:=FALSE;END_IF
IF NOT LotAHmi AND NOT LotBHmi AND  LotCHmi THEN LotCSelected:=TRUE;LotBSelected:=FALSE;LotASelected:=FALSE;END_IF

IF LotASelected THEN CartonNoHmi:=LotACartonNo;
ELSIF LotBSelected THEN CartonNoHmi:=LotBCartonNo;
ELSIF  LotCSelected THEN CartonNoHmi:=LotCCartonNo;
ELSIF  LotDSelected THEN CartonNoHmi:=LotDCartonNo;
ELSIF  LotESelected THEN CartonNoHmi:=LotECartonNo;
ELSIF  LotFSelected THEN CartonNoHmi:=LotFCartonNo;
END_IF

IF CartonNoResetHmi OR  (NOT LotAHmi AND NOT LotBHmi AND NOT LotCHmi) THEN
	LotACartonNo:=0;
	LotBCartonNo:=0;
	LotCCartonNo:=0;
	LotDCartonNo:=0;
	LotECartonNo:=0;
	LotFCartonNo:=0;
END_IF



CASE LotA OF

0:	IF LotASelected THEN LotA:=LotA+1;END_IF

1:	IF (CycleComplete OR CycleComplete1) THEN LotA :=LotA +1;END_IF

2:	LotACartonNo:=LotACartonNo+1;
	LotA :=LotA +1;

3:	TON_11(IN:=TRUE , PT:=t#25s , Q=> , ET=> );
	IF TON_11.Q THEN LotA :=LotA +1;END_IF

4:	LotA :=0;

END_CASE


CASE LotB OF

0:	IF LotBSelected THEN LotB:=LotB+1;END_IF

1:	IF (CycleComplete OR CycleComplete1) THEN LotB:=LotB+1;END_IF

2:	LotBCartonNo:=LotBCartonNo+1;
	LotB:=LotB+1;

3:	TON_12(IN:=TRUE , PT:=t#25s , Q=> , ET=> );
	IF TON_12.Q THEN LotA :=LotA +1;END_IF

4:	LotB:=0;

END_CASE


CASE LotC OF

0:	IF LotCSelected THEN LotC:=LotC+1;END_IF

1:	IF (CycleComplete OR CycleComplete1) THEN LotC:=LotC+1;END_IF

2:	LotCCartonNo:=LotCCartonNo+1;
	LotC:=LotC+1;

3:	TON_13(IN:=TRUE , PT:=t#25s , Q=> , ET=> );
	IF TON_13.Q THEN LotA :=LotA +1;END_IF

4:	LotC:=0;

END_CASE*)*)
END_PROGRAM

(* POU FunctionBlocks/DATA_LOG_Save, ST *)
FUNCTION_BLOCK DATA_LOG_Save
VAR_INPUT
	bStartDataLog: BOOL;
	sDataLogFileName: STRING;
	LogData: STRING(1024);

END_VAR
VAR_OUTPUT

	bErrorDataLog: BOOL;
END_VAR
VAR

	R_TRIGStartDataLog: R_TRIG;
	nstep: INT;

	FB_OpenFile_Datalog: FB_FileOpen;
	nFB_OpenFile_Datalog_Errid: UDINT;

	FB_WriteFile_Datalog: FB_FileWrite;
	nFB_WriteFile_Datalog_ErrId: UDINT;

	FB_CloseFile_Datalog: FB_FileClose;
	nFB_CloseFile_Datalog_ErrId: UDINT;
	hDataLogSrcFile: UINT;

END_VAR
;(*R_TRIGStartDataLog(CLK:=bStartDataLog , Q=> );
IF R_TRIGStartDataLog.Q THEN
		nstep :=1;
	END_IF

CASE nstep OF

	0:
		;
		FB_OpenFile_Datalog.bExecute:=FALSE;
		FB_WriteFile_Datalog.bExecute:=FALSE;
		FB_CloseFile_Datalog.bExecute:=FALSE;

	1:		(* do nothing *)
			nstep:=nstep+1;

	2:		(* ####	File Open ####*)

			FB_OpenFile_Datalog(  bExecute := FALSE  );
			FB_OpenFile_Datalog(	sNetId :='192.168.0.103.1.1' ,
			sPathName := sDataLogFileName,
			nMode := FOPEN_MODEAPPEND    ,
			ePath := PATH_GENERIC,
			tTimeout := T#2s,
			bExecute := TRUE );
			nstep := nstep+ 1;



	3:		FB_OpenFile_Datalog( bExecute := FALSE );
			IF ( NOT FB_OpenFile_Datalog.bBusy ) THEN
			IF ( FB_OpenFile_Datalog.bError ) THEN
			nFB_OpenFile_Datalog_Errid := FB_OpenFile_Datalog.nErrId;
			bErrorDataLog := TRUE;
			nstep := 50;
			ELSE
			hDataLogSrcFile := FB_OpenFile_Datalog.hFile;
			nstep := nstep + 1;
			END_IF
			END_IF

	4:		(*write data to destination file*)
			(*num:=num+1;*)
			FB_WriteFile_Datalog( bExecute := FALSE );
			FB_WriteFile_Datalog(	sNetId:='192.168.0.103.1.1',
			hFile:=FB_OpenFile_Datalog.hFile,
			pWriteBuff:= ADR(LogData),
			cbWriteLen:= LEN(LogData),		(*	i_len,	*)
			bExecute:=TRUE,
			tTimeout:=T#2s );
			nstep := nstep + 1;

	5:		FB_WriteFile_Datalog( bExecute := FALSE );
			IF ( NOT FB_WriteFile_Datalog.bBusy ) THEN
			IF ( FB_WriteFile_Datalog.bError ) THEN
			nFB_WriteFile_Datalog_ErrId := FB_WriteFile_Datalog.nErrId;
			bErrorDataLog := TRUE;
			nstep := 50;
			ELSE
			hDataLogSrcFile := FB_OpenFile_Datalog.hFile;
			nstep := nstep + 1;
			END_IF
			END_IF

	6:		(* close the destination file *)
			FB_CloseFile_Datalog( bExecute := FALSE );
			FB_CloseFile_Datalog( 	sNetId:='192.168.0.103.1.1' ,
			hFile:=FB_OpenFile_Datalog.hFile,
			bExecute:=TRUE,
			tTimeout:=T#2s );
			nstep := nstep + 1;

	7:		FB_CloseFile_Datalog( bExecute := FALSE );
			IF ( NOT FB_CloseFile_Datalog.bBusy ) THEN
			IF ( FB_CloseFile_Datalog.bError ) THEN
			nFB_CloseFile_Datalog_ErrId := FB_CloseFile_Datalog.nErrId;
			bErrorDataLog := TRUE;
			END_IF
			nstep := 0;
			END_IF

END_CASE*)
END_FUNCTION_BLOCK

(* POU FunctionBlocks/Fb_CreateFileFormat, LD *)
FUNCTION_BLOCK Fb_CreateFileFormat
VAR
	Fb_OpenFile: FB_FileOpen;
	Fb_WriteFile: FB_FileWrite;
	F_Trig1: F_TRIG;
	F_Trig2: F_TRIG;
	Fb_closeFile: FB_FileClose;
	F_Trig3: F_TRIG;


	SysteMtime: FB_LocalSystemTime;
	stSystemtimeAlrm: Timestruct;

	sFileName_Temp: T_MaxString;


	bCreateFileTrig: R_TRIG;
	bCreateFile: BOOL;
	Fb_SavePersistant: FB_WritePersistentData;
	TuneparaSave: BOOL;
END_VAR
VAR_INPUT

	sInputMessage: STRING(255);
	sFileName: T_MaxString;
	sDirectory: T_MaxString;
	bEnable: BOOL;

END_VAR
VAR_OUTPUT

	sDate: STRING;

	bNewDateFound: BOOL;
END_VAR

VAR_OUTPUT PERSISTENT
	sOldFileName: T_MaxString;
	sFilePathFinal: t_MaxString;
END_VAR
VAR PERSISTENT
	sOldDate: STRING;
	sNewFileName_Temp: T_MaxString;
END_VAR
VAR_IN_OUT PERSISTENT
	wToday: STRING;
END_VAR
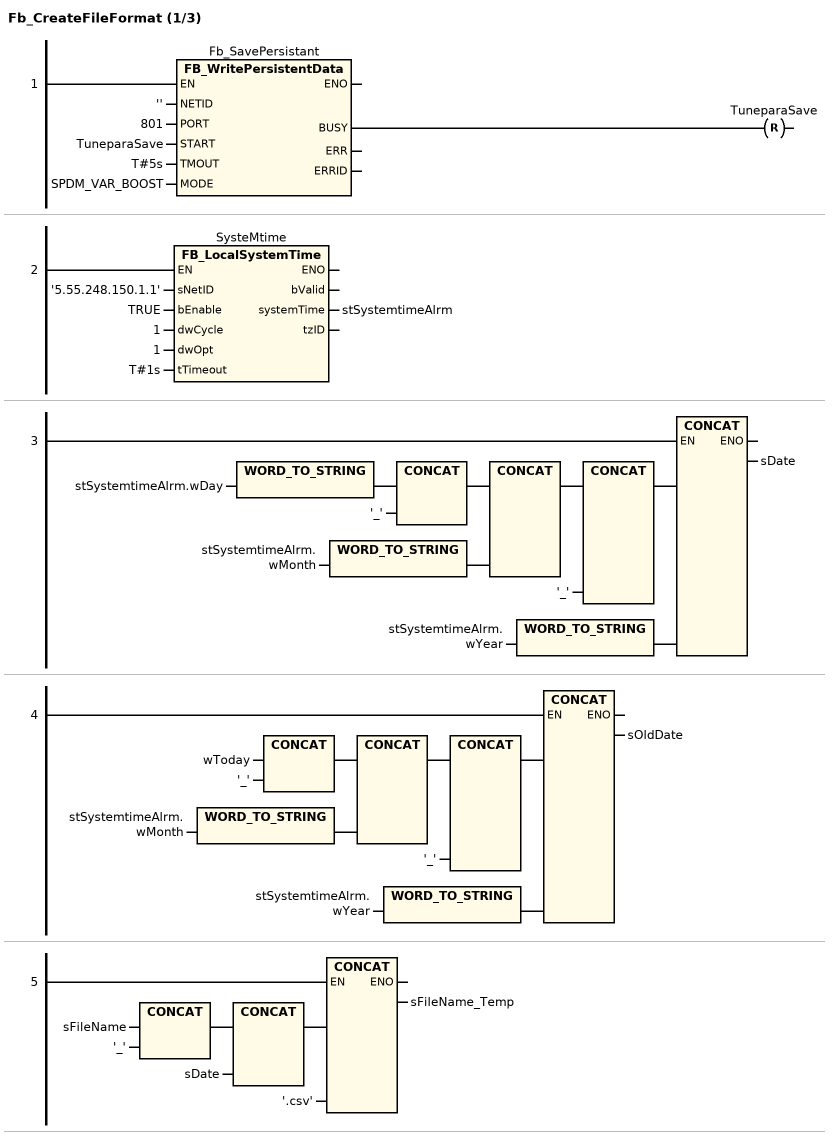
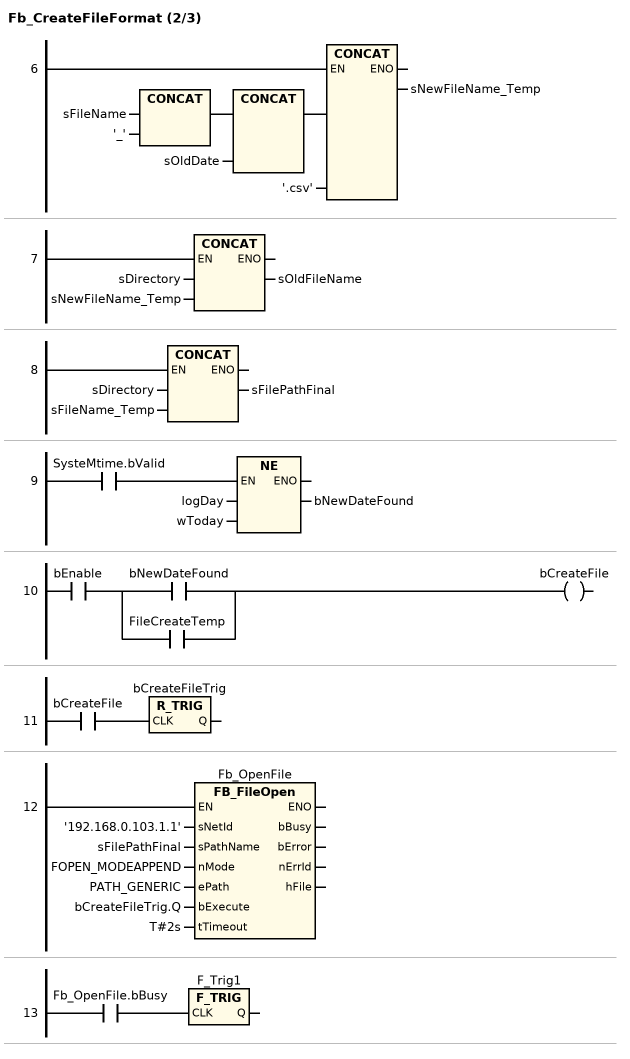
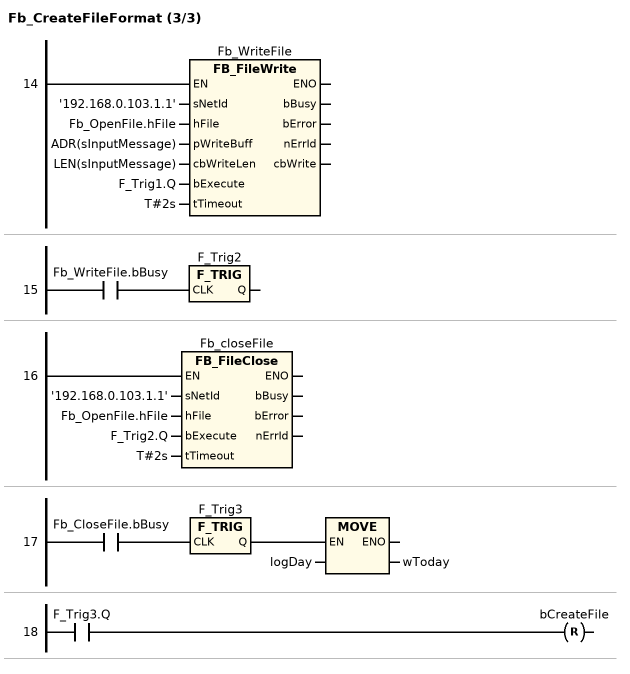
_LD_ (* Ladder Diagram *)
NETWORK 1
	*
		EN --- Fb_SavePersistant:FB_WritePersistentData(NETID: '', PORT: 801, START: TuneparaSave, TMOUT: T#5s, MODE: SPDM_VAR_BOOST) => R TuneparaSave
NETWORK 2
	*
		EN --- SysteMtime:FB_LocalSystemTime(sNetID: '5.55.248.150.1.1', bEnable: TRUE, dwCycle: 1, dwOpt: 1, tTimeout: T#1s, systemTime => stSystemtimeAlrm)
NETWORK 3
	*
		EN --- CONCAT(CONCAT(CONCAT(CONCAT(WORD_TO_STRING(stSystemtimeAlrm.wDay), '_'), WORD_TO_STRING(stSystemtimeAlrm.wMonth)), '_'), WORD_TO_STRING(stSystemtimeAlrm.wYear)) => sDate
NETWORK 4
	*
		EN --- CONCAT(CONCAT(CONCAT(CONCAT(wToday, '_'), WORD_TO_STRING(stSystemtimeAlrm.wMonth)), '_'), WORD_TO_STRING(stSystemtimeAlrm.wYear)) => sOldDate
NETWORK 5
	*
		EN --- CONCAT(CONCAT(CONCAT(sFileName, '_'), sDate), '.csv') => sFileName_Temp
NETWORK 6
	*
		EN --- CONCAT(CONCAT(CONCAT(sFileName, '_'), sOldDate), '.csv') => sNewFileName_Temp
NETWORK 7
	*
		EN --- CONCAT(sDirectory, sNewFileName_Temp) => sOldFileName
NETWORK 8
	*
		EN --- CONCAT(sDirectory, sFileName_Temp) => sFilePathFinal
NETWORK 9
	[SysteMtime.bValid]
		EN --- NE(logDay, wToday) => bNewDateFound
NETWORK 10
	[bEnable] - { [bNewDateFound] | [FileCreateTemp] } --- (bCreateFile)
NETWORK 11
	[bCreateFile] - bCreateFileTrig:R_TRIG(CLK: *)
NETWORK 12
	*
		EN --- Fb_OpenFile:FB_FileOpen(sNetId: '192.168.0.103.1.1', sPathName: sFilePathFinal, nMode: FOPEN_MODEAPPEND, ePath: PATH_GENERIC, bExecute: bCreateFileTrig.Q, tTimeout: T#2s)
NETWORK 13
	[Fb_OpenFile.bBusy] - F_Trig1:F_TRIG(CLK: *)
NETWORK 14
	*
		EN --- Fb_WriteFile:FB_FileWrite(sNetId: '192.168.0.103.1.1', hFile: Fb_OpenFile.hFile, pWriteBuff: ADR(sInputMessage), cbWriteLen: LEN(sInputMessage), bExecute: F_Trig1.Q, tTimeout: T#2s)
NETWORK 15
	[Fb_WriteFile.bBusy] - F_Trig2:F_TRIG(CLK: *)
NETWORK 16
	*
		EN --- Fb_closeFile:FB_FileClose(sNetId: '192.168.0.103.1.1', hFile: Fb_OpenFile.hFile, bExecute: F_Trig2.Q, tTimeout: T#2s)
NETWORK 17
	[Fb_CloseFile.bBusy] - F_Trig3:F_TRIG(CLK: *)
		EN --- MOVE(logDay) => wToday
NETWORK 18
	[F_Trig3.Q] --- (R bCreateFile)
_END_LD_
(* the same logic as Structured Text *)
(* Network 1 *)
Fb_SavePersistant(NETID := '', PORT := 801, START := TuneparaSave, TMOUT := T#5s, MODE := SPDM_VAR_BOOST);
IF Fb_SavePersistant.BUSY THEN TuneparaSave := FALSE; END_IF;
(* Network 2 *)
SysteMtime(sNetID := '5.55.248.150.1.1', bEnable := TRUE, dwCycle := 1, dwOpt := 1, tTimeout := T#1s);
stSystemtimeAlrm := SysteMtime.systemTime;
(* Network 3 *)
sDate := CONCAT(CONCAT(CONCAT(CONCAT(WORD_TO_STRING(stSystemtimeAlrm.wDay), '_'), WORD_TO_STRING(stSystemtimeAlrm.wMonth)), '_'), WORD_TO_STRING(stSystemtimeAlrm.wYear));
(* Network 4 *)
sOldDate := CONCAT(CONCAT(CONCAT(CONCAT(wToday, '_'), WORD_TO_STRING(stSystemtimeAlrm.wMonth)), '_'), WORD_TO_STRING(stSystemtimeAlrm.wYear));
(* Network 5 *)
sFileName_Temp := CONCAT(CONCAT(CONCAT(sFileName, '_'), sDate), '.csv');
(* Network 6 *)
sNewFileName_Temp := CONCAT(CONCAT(CONCAT(sFileName, '_'), sOldDate), '.csv');
(* Network 7 *)
sOldFileName := CONCAT(sDirectory, sNewFileName_Temp);
(* Network 8 *)
sFilePathFinal := CONCAT(sDirectory, sFileName_Temp);
(* Network 9 *)
IF SysteMtime.bValid THEN
	bNewDateFound := logDay <> wToday;
END_IF;
(* Network 10 *)
bCreateFile := bEnable AND (bNewDateFound OR FileCreateTemp);
(* Network 11 *)
bCreateFileTrig(CLK := bCreateFile);
(* Network 12 *)
Fb_OpenFile(sNetId := '192.168.0.103.1.1', sPathName := sFilePathFinal, nMode := FOPEN_MODEAPPEND, ePath := PATH_GENERIC, bExecute := bCreateFileTrig.Q, tTimeout := T#2s);
(* Network 13 *)
F_Trig1(CLK := Fb_OpenFile.bBusy);
(* Network 14 *)
Fb_WriteFile(sNetId := '192.168.0.103.1.1', hFile := Fb_OpenFile.hFile, pWriteBuff := ADR(sInputMessage), cbWriteLen := LEN(sInputMessage), bExecute := F_Trig1.Q, tTimeout := T#2s);
(* Network 15 *)
F_Trig2(CLK := Fb_WriteFile.bBusy);
(* Network 16 *)
Fb_closeFile(sNetId := '192.168.0.103.1.1', hFile := Fb_OpenFile.hFile, bExecute := F_Trig2.Q, tTimeout := T#2s);
(* Network 17 *)
F_Trig3(CLK := Fb_CloseFile.bBusy);
IF F_Trig3.Q THEN
	wToday := logDay;
END_IF;
(* Network 18 *)
IF F_Trig3.Q THEN bCreateFile := FALSE; END_IF;
END_FUNCTION_BLOCK

(* POU FunctionBlocks/Fb_FormatDrive, FBD *)
FUNCTION_BLOCK Fb_FormatDrive
VAR_INPUT
	sDriveName: T_MaxString;
	bFormatDisk: BOOL;
END_VAR
VAR_OUTPUT
END_VAR
VAR
	sDeleteCommand_Temp: T_MaxString;
	sDeleteCommand: T_MaxString;
	nDirectoryLength: INT;
	sFormatedDirectory: T_MaxString;
	FbFormatDisk: NT_StartProcess;
END_VAR
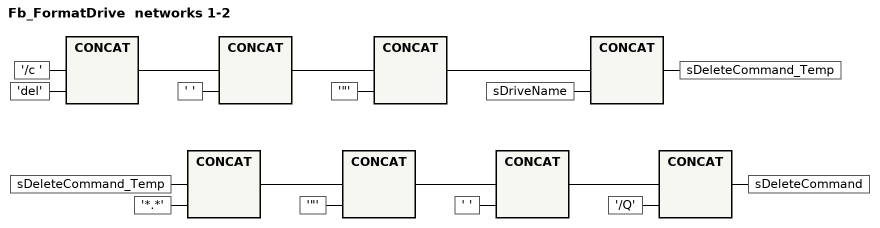
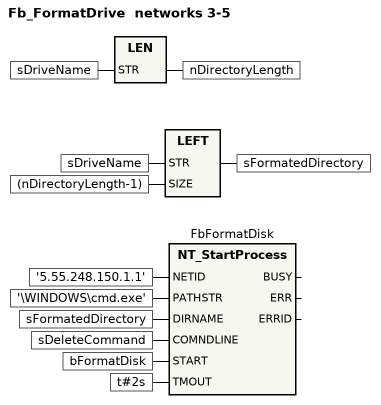
_FBD_ (* Function Block Diagram *)
NETWORK 1
	CONCAT(CONCAT(CONCAT(CONCAT('/c ', 'del'), ' '), '"'), sDriveName) => sDeleteCommand_Temp
NETWORK 2
	CONCAT(CONCAT(CONCAT(CONCAT(sDeleteCommand_Temp, '*.*'), '"'), ' '), '/Q') => sDeleteCommand
NETWORK 3
	LEN(STR: sDriveName) => nDirectoryLength
NETWORK 4
	LEFT(STR: sDriveName, SIZE: (nDirectoryLength-1)) => sFormatedDirectory
NETWORK 5
	FbFormatDisk:NT_StartProcess(NETID: '5.55.248.150.1.1', PATHSTR: '\WINDOWS\cmd.exe', DIRNAME: sFormatedDirectory, COMNDLINE: sDeleteCommand, START: bFormatDisk, TMOUT: t#2s)
_END_FBD_
(* the same logic as Structured Text *)
(* Network 1 *)
sDeleteCommand_Temp := CONCAT(CONCAT(CONCAT(CONCAT('/c ', 'del'), ' '), '"'), sDriveName);
(* Network 2 *)
sDeleteCommand := CONCAT(CONCAT(CONCAT(CONCAT(sDeleteCommand_Temp, '*.*'), '"'), ' '), '/Q');
(* Network 3 *)
nDirectoryLength := LEN(sDriveName);
(* Network 4 *)
sFormatedDirectory := LEFT(sDriveName, (nDirectoryLength-1));
(* Network 5 *)
FbFormatDisk(NETID := '5.55.248.150.1.1', PATHSTR := '\WINDOWS\cmd.exe', DIRNAME := sFormatedDirectory, COMNDLINE := sDeleteCommand, START := bFormatDisk, TMOUT := t#2s);
END_FUNCTION_BLOCK

(* POU FunctionBlocks/Fb_CopyFileToRemotePC, FBD *)
FUNCTION_BLOCK Fb_CopyFileToRemotePC
VAR
	sCopyFileCommandTemp: T_MaxString;
	sFormatedDestDirectory: T_Maxstring;
	sCopyFileCommand: T_MaxString;
	sFormatedDirectory: T_MaxString;
	sMakeDirCommand: T_MaxString;

	Fb_SystemTime: FB_LocalSystemTime;
	FB_MakeDirectory: NT_StartProcess;
	Fb_CopyFiles: NT_StartProcess;
END_VAR
VAR_INPUT

	bMakeDirectory: BOOL;
	bCopyFile: BOOL;
	sDestDriveName: T_MaxString;
	sSourceDirectory: T_MaxString;
END_VAR
VAR_OUTPUT
	sFinalDestDirectory: T_MaxString;
END_VAR
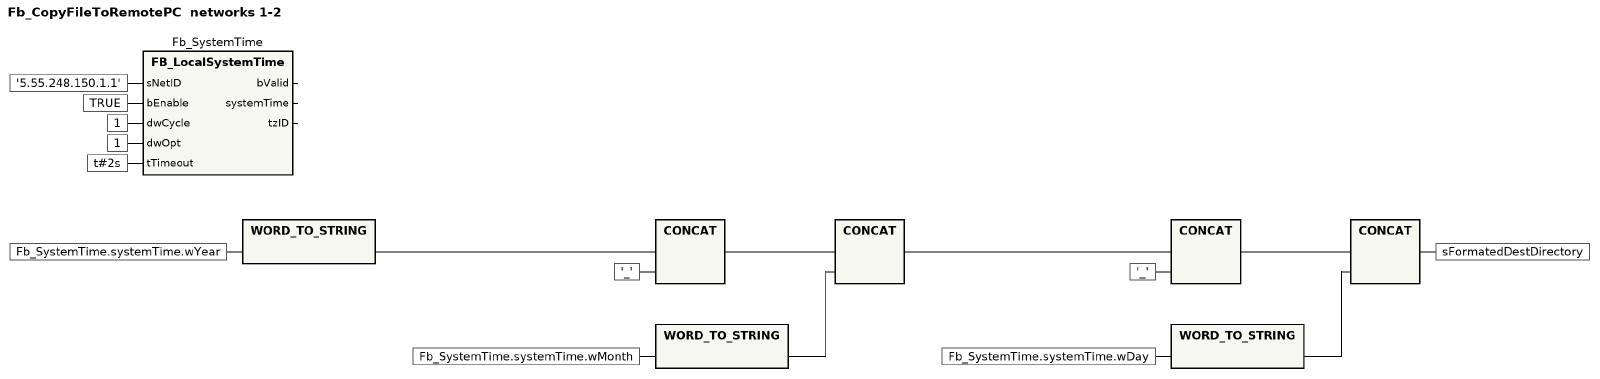
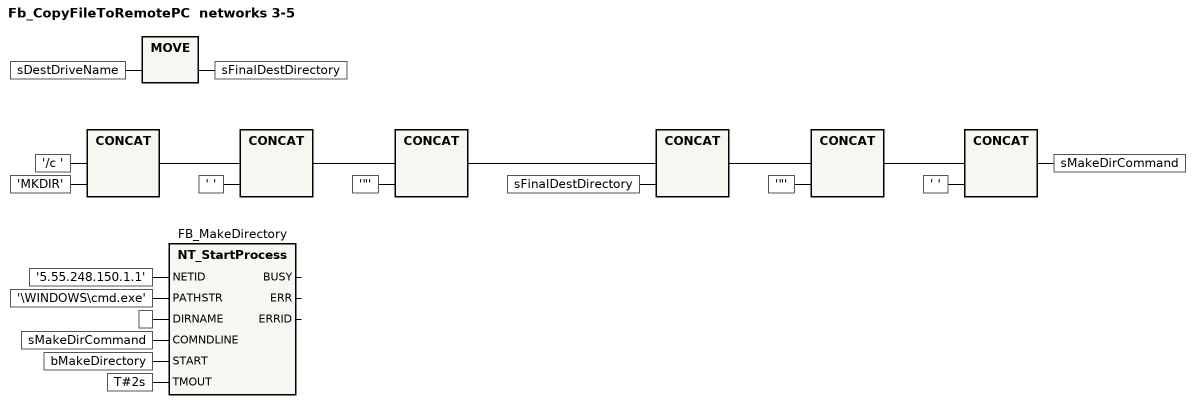
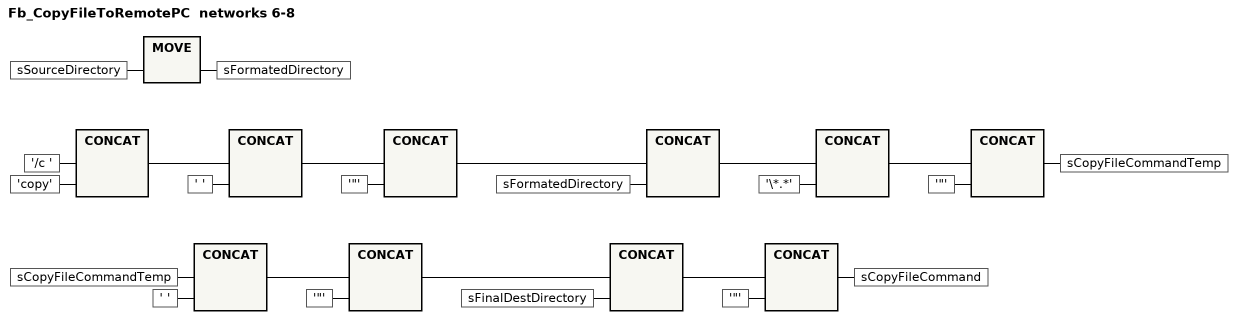
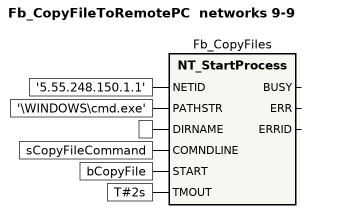
_FBD_ (* Function Block Diagram *)
NETWORK 1
	Fb_SystemTime:FB_LocalSystemTime(sNetID: '5.55.248.150.1.1', bEnable: TRUE, dwCycle: 1, dwOpt: 1, tTimeout: t#2s)
NETWORK 2
	CONCAT(CONCAT(CONCAT(CONCAT(WORD_TO_STRING(Fb_SystemTime.systemTime.wYear), '_'), WORD_TO_STRING(Fb_SystemTime.systemTime.wMonth)), '_'), WORD_TO_STRING(Fb_SystemTime.systemTime.wDay)) => sFormatedDestDirectory
NETWORK 3
	MOVE(sDestDriveName) => sFinalDestDirectory
NETWORK 4
	CONCAT(CONCAT(CONCAT(CONCAT(CONCAT(CONCAT('/c ', 'MKDIR'), ' '), '"'), sFinalDestDirectory), '"'), ' ') => sMakeDirCommand
NETWORK 5
	FB_MakeDirectory:NT_StartProcess(NETID: '5.55.248.150.1.1', PATHSTR: '\WINDOWS\cmd.exe', DIRNAME: , COMNDLINE: sMakeDirCommand, START: bMakeDirectory, TMOUT: T#2s)
NETWORK 6
	MOVE(sSourceDirectory) => sFormatedDirectory
NETWORK 7
	CONCAT(CONCAT(CONCAT(CONCAT(CONCAT(CONCAT('/c ', 'copy'), ' '), '"'), sFormatedDirectory), '\*.*'), '"') => sCopyFileCommandTemp
NETWORK 8
	CONCAT(CONCAT(CONCAT(CONCAT(sCopyFileCommandTemp, ' '), '"'), sFinalDestDirectory), '"') => sCopyFileCommand
NETWORK 9
	Fb_CopyFiles:NT_StartProcess(NETID: '5.55.248.150.1.1', PATHSTR: '\WINDOWS\cmd.exe', DIRNAME: , COMNDLINE: sCopyFileCommand, START: bCopyFile, TMOUT: T#2s)
_END_FBD_
(* the same logic as Structured Text *)
(* Network 1 *)
Fb_SystemTime(sNetID := '5.55.248.150.1.1', bEnable := TRUE, dwCycle := 1, dwOpt := 1, tTimeout := t#2s);
(* Network 2 *)
sFormatedDestDirectory := CONCAT(CONCAT(CONCAT(CONCAT(WORD_TO_STRING(Fb_SystemTime.systemTime.wYear), '_'), WORD_TO_STRING(Fb_SystemTime.systemTime.wMonth)), '_'), WORD_TO_STRING(Fb_SystemTime.systemTime.wDay));
(* Network 3 *)
sFinalDestDirectory := sDestDriveName;
(* Network 4 *)
sMakeDirCommand := CONCAT(CONCAT(CONCAT(CONCAT(CONCAT(CONCAT('/c ', 'MKDIR'), ' '), '"'), sFinalDestDirectory), '"'), ' ');
(* Network 5: see the listing above *)
(* Network 6 *)
sFormatedDirectory := sSourceDirectory;
(* Network 7 *)
sCopyFileCommandTemp := CONCAT(CONCAT(CONCAT(CONCAT(CONCAT(CONCAT('/c ', 'copy'), ' '), '"'), sFormatedDirectory), '\*.*'), '"');
(* Network 8 *)
sCopyFileCommand := CONCAT(CONCAT(CONCAT(CONCAT(sCopyFileCommandTemp, ' '), '"'), sFinalDestDirectory), '"');
(* Network 9: see the listing above *)
END_FUNCTION_BLOCK

(* Visualisation A
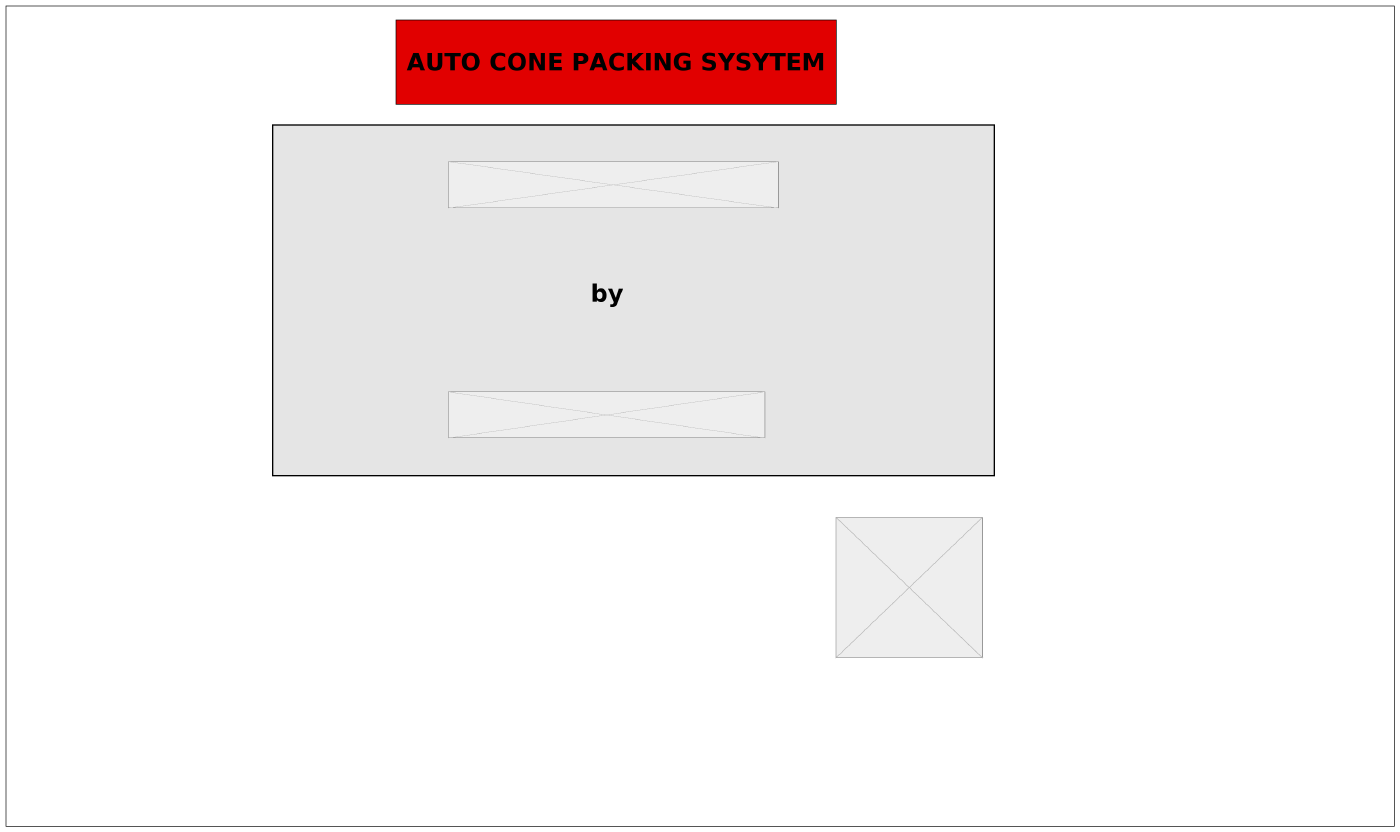
group at (380,20)-(1411,931)
  rounded rectangle at (144,0)-(657,97): text "AUTO CONE PACKING SYSYTEM"
  bitmap at (656,568)-(827,729): c:\twincat\plc\visu\startbutton.jpg
  group at (0,120)-(841,521)
    rounded rectangle at (0,0)-(1051,611): invisible if Common.EverRunTimer.Q
    bitmap at (256,64)-(737,145): c:\twincat\plc\visu\autocone-logom1.jpg
    bitmap at (256,464)-(717,545): c:\twincat\plc\visu\indo_logo1.bmp
    rectangle at (232,248)-(743,339): text "by"
2 more shapes without text or variables
*)

(* Visualisation ALARM
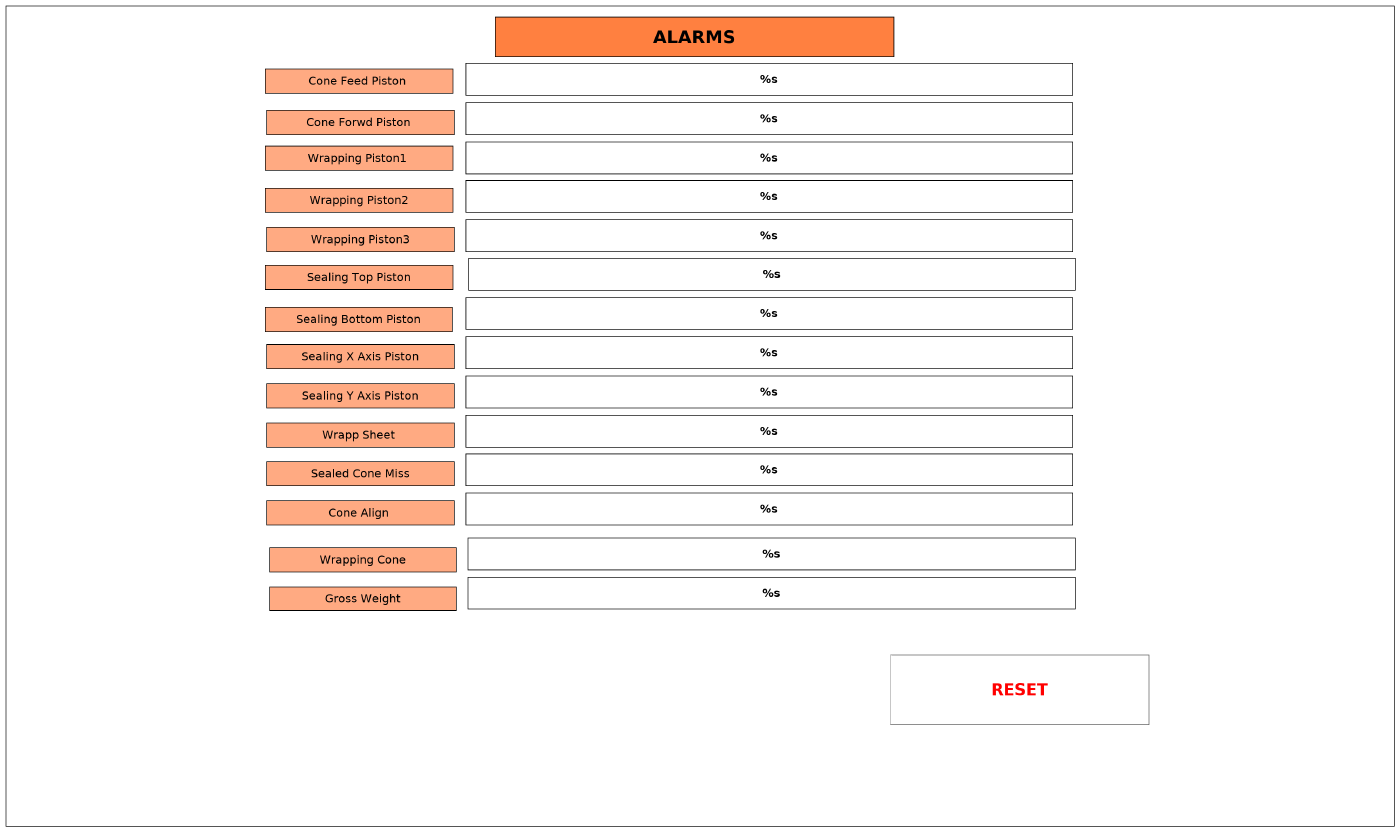
rounded rectangle at (372,149)-(640,184): text "Cone Forwd Piston"
rounded rectangle at (370,90)-(638,125): text "Cone Feed Piston"
rounded rectangle at (370,200)-(638,235): text "Wrapping Piston1"
rounded rectangle at (370,260)-(638,295): text "Wrapping Piston2"
rounded rectangle at (372,316)-(640,351): text "Wrapping Piston3"
rounded rectangle at (370,370)-(638,405): text "Sealing Top Piston"
rounded rectangle at (370,430)-(637,465): text "Sealing Bottom Piston"
rounded rectangle at (372,483)-(640,518): text "Sealing X Axis Piston"
rounded rectangle at (372,539)-(640,574): text "Sealing Y Axis Piston"
rectangle at (656,82)-(1522,128): text "%s"; shows .HMIFeedPiston
rectangle at (656,305)-(1522,351): text "%s"; shows .HMIWrapPiston3
rectangle at (656,249)-(1522,295): text "%s"; shows .HMIWrapPiston2
rectangle at (660,360)-(1526,406): text "%s"; shows .HMISealTopPiston
rectangle at (656,472)-(1522,518): text "%s"; shows .HmiXAxisPiston
rectangle at (656,416)-(1522,462): text "%s"; shows .HMISealBotPiston
rectangle at (656,528)-(1522,574): text "%s"; shows .HmiYAxisPiston
rectangle at (656,194)-(1522,240): text "%s"; shows .HMIWrapPiston1
rectangle at (656,138)-(1522,184): text "%s"; shows .HMIForwdPiston
button at (1262,926)-(1631,1026): text "RESET"; shows .bErrorResethmi; taps .bErrorResethmi
rounded rectangle at (372,595)-(640,630): text "Wrapp Sheet"
rectangle at (656,584)-(1522,630): text "%s"; shows ConeMissAlarm1
rounded rectangle at (372,650)-(640,685): text "Sealed Cone Miss"
rectangle at (656,639)-(1522,685): text "%s"; shows .AlarmMessg
rounded rectangle at (372,706)-(640,741): text "Cone Align"
rectangle at (656,695)-(1522,741): text "%s"; shows .ConeMissAlarm
rounded rectangle at (698,16)-(1267,73): text "ALARMS"
rectangle at (659,759)-(1526,805): text "%s"; shows WrapConeSenDetMes
rounded rectangle at (376,773)-(643,808): text "Wrapping Cone"
rectangle at (659,815)-(1526,861): text "%s"; shows SGrossWtNokMsg
rounded rectangle at (376,829)-(643,863): text "Gross Weight"
1 more shapes without text or variables
2 elements of other kinds (tables, trends, ...) not read
*)

(* Visualisation ALARM_2
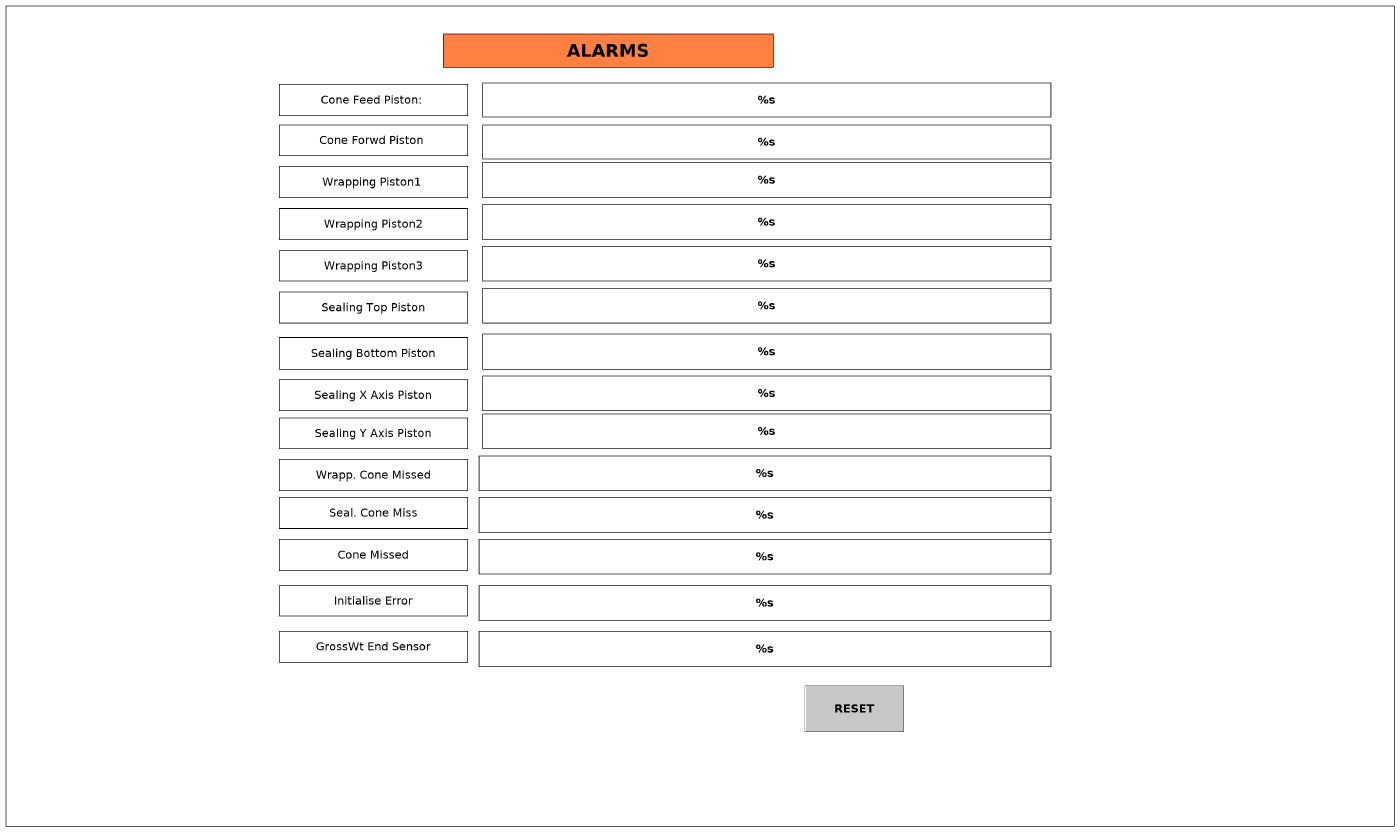
button at (1140,970)-(1281,1036): text "RESET"; shows .bErrorResethmi; taps .bErrorResethmi
rounded rectangle at (624,40)-(1095,88): text "ALARMS"
rounded rectangle at (390,170)-(659,214): text "Cone Forwd Piston"
rounded rectangle at (390,112)-(659,157): text "Cone Feed Piston:"
rounded rectangle at (390,229)-(659,274): text "Wrapping Piston1"
rounded rectangle at (390,289)-(659,334): text "Wrapping Piston2"
rounded rectangle at (390,349)-(659,393): text "Wrapping Piston3"
rounded rectangle at (390,408)-(659,453): text "Sealing Top Piston"
rounded rectangle at (390,473)-(659,519): text "Sealing Bottom Piston"
rounded rectangle at (390,533)-(659,578): text "Sealing X Axis Piston"
rounded rectangle at (390,588)-(659,632): text "Sealing Y Axis Piston"
rectangle at (680,110)-(1491,159): text "%s"; shows .HMIFeedPiston
rectangle at (680,343)-(1491,393): text "%s"; shows .HMIWrapPiston3
rectangle at (680,283)-(1491,334): text "%s"; shows .HMIWrapPiston2
rectangle at (680,403)-(1491,453): text "%s"; shows .HMISealTopPiston
rectangle at (680,528)-(1491,578): text "%s"; shows .HmiXAxisPiston
rectangle at (680,468)-(1491,519): text "%s"; shows .HMISealBotPiston
rectangle at (680,582)-(1491,632): text "%s"; shows .HmiYAxisPiston
rectangle at (680,223)-(1491,274): text "%s"; shows .HMIWrapPiston1
rectangle at (680,170)-(1491,219): text "%s"; shows .HMIForwdPiston
rounded rectangle at (390,647)-(659,692): text "Wrapp. Cone Missed"
rectangle at (675,642)-(1491,692): text "%s"; shows .ConeMissAlarm
rounded rectangle at (390,701)-(659,746): text "Seal. Cone Miss"
rectangle at (675,701)-(1491,752): text "%s"; shows .AlarmMessg
rounded rectangle at (390,761)-(659,806): text "Cone Missed"
rectangle at (675,761)-(1491,811): text "%s"; shows .ConeMissAlarm
rounded rectangle at (390,827)-(659,871): text "Initialise Error"
rectangle at (675,827)-(1491,877): text "%s"; shows sMessage
rounded rectangle at (390,892)-(659,937): text "GrossWt End Sensor"
rectangle at (675,892)-(1491,943): text "%s"; shows SGrossWtCylEndSenErrMsg
1 more shapes without text or variables
2 elements of other kinds (tables, trends, ...) not read
*)

